 (*Zachowanie po stopie awaryjnym*)
 IF P00_Alarms.aLastStationsErrors[1].nErrorCode >= 1 AND P00_Alarms.aLastStationsErrors[1].nErrorCode <= 20 THEN
     //Jezeli było w trakcie dozowania i coś wydozowało
     IF (iDispencersCase = 4 ) OR (lrDosedMass1CVAux>2 OR lrDosedMass2CVAux>2 OR lrDosedMass3CVAux>2 OR lrDosedMass4CVAux > 2) THEN
         eDispencersPackageState[4].bDoseAborted:=TRUE;
         eDispencersPackageState[3].bDoseAborted:=TRUE;
         eDispencersPackageState[2].bDoseAborted:=TRUE;
         eDispencersPackageState[1].bDoseAborted:=TRUE;
     END_IF
 END_IF
 (*Zachowanie po jakimkolwiek błędzie dozownika 1 i dozownika 2*)
 IF P00_Alarms.aLastStationsErrors[9].bError OR P00_Alarms.aLastStationsErrors[10].bError OR P00_Alarms.aLastStationsErrors[11].bError OR P00_Alarms.aLastStationsErrors[12].bError  THEN
     //Jezeli było w trakcie dozowania i coś wydozowało
     IF (iDispencersCase = 4 ) OR (ABS(lrDosedMass1CVAux)>2 OR ABS(lrDosedMass2CVAux)>2 OR ABS(lrDosedMass3CVAux)>2 OR ABS(lrDosedMass4CVAux) > 2) THEN
         eDispencersPackageState[4].bDoseAborted:=TRUE;
         eDispencersPackageState[3].bDoseAborted:=TRUE;
         eDispencersPackageState[2].bDoseAborted:=TRUE;
         eDispencersPackageState[1].bDoseAborted:=TRUE;
     END_IF
 END_IF
  (*Zachowanie po błędzie przeciagania*)
 IF P00_Alarms.aLastStationsErrors[4].bError OR P00_Alarms.aLastStationsErrors[41].bError OR (P00_Alarms.aLastStationsErrors[1].bError AND P00_Alarms.aLastStationsErrors[1].nErrorCode=70)THEN //Prawe/Lewe
         eBeforeDispencersPackageState[4].bDoseAborted:=TRUE;
         eBeforeDispencersPackageState[3].bDoseAborted:=TRUE;
         eBeforeDispencersPackageState[2].bDoseAborted:=TRUE;
         eBeforeDispencersPackageState[1].bDoseAborted:=TRUE;
     	 eDispencersPackageState[4].bDoseAborted:=TRUE;
         eDispencersPackageState[3].bDoseAborted:=TRUE;
         eDispencersPackageState[2].bDoseAborted:=TRUE;
         eDispencersPackageState[1].bDoseAborted:=TRUE;		  
 END_IF
 
(*Zachowanie po błędzie sortera nasadek*)
 IF P00_Alarms.aLastStationsErrors[50].bError THEN
	
		iCapSorterCase := 0;
		eCapSorterPackageState[1].bCapSorterPuttedAborted	:=	TRUE;
		eCapSorterPackageState[2].bCapSorterPuttedAborted	:=	TRUE;
		eCapSorterPackageState[3].bCapSorterPuttedAborted	:=	TRUE;
		eCapSorterPackageState[4].bCapSorterPuttedAborted	:=	TRUE;
	
 END_IF
 
 (*
 (*Zachowanie po błędzie przeciągania sortera nasadek*)	(*Błąd zablokowanej nasadki*)
 IF P00_Alarms.aLastStationsErrors[51].bError OR (P00_Alarms.aLastStationsErrors[1].bError AND P00_Alarms.aLastStationsErrors[1].nErrorCode=64) THEN
	
		eCapSorterPackageState[1].bCapSorterPuttedAborted	:=	TRUE;
		eCapSorterPackageState[2].bCapSorterPuttedAborted	:=	TRUE;
		eCapSorterPackageState[3].bCapSorterPuttedAborted	:=	TRUE;
		eCapSorterPackageState[4].bCapSorterPuttedAborted	:=	TRUE;

		eBeforeCapSorterPackageState[1].bCapSorterPuttedAborted	:=	TRUE;
		eBeforeCapSorterPackageState[2].bCapSorterPuttedAborted	:=	TRUE;
		eBeforeCapSorterPackageState[3].bCapSorterPuttedAborted	:=	TRUE;
		eBeforeCapSorterPackageState[4].bCapSorterPuttedAborted	:=	TRUE;
	
 END_IF
 *)
END_ACTION

ACTION ACT_ResetAfterStart:
	IF rtResetAfterStart.Q THEN //po 60s
		
		GVL.eCapSorterPackageState[1] 				:= GVL.eClearPackageState;
		GVL.eCapSorterPackageState[2] 				:= GVL.eClearPackageState;
		GVL.eCapSorterPackageState[3] 				:= GVL.eClearPackageState;
		GVL.eCapSorterPackageState[4] 				:= GVL.eClearPackageState;	
	
		GVL.eBeforeCapSorterPackageState[1] 		:= GVL.eClearPackageState;
		GVL.eBeforeCapSorterPackageState[2] 		:= GVL.eClearPackageState;
		GVL.eBeforeCapSorterPackageState[3] 		:= GVL.eClearPackageState;
		GVL.eBeforeCapSorterPackageState[4] 		:= GVL.eClearPackageState;
	
		GVL.eWeightPackageState[1] 					:= GVL.eClearPackageState;
		GVL.eWeightPackageState[2] 					:= GVL.eClearPackageState;
		GVL.eWeightPackageState[3] 					:= GVL.eClearPackageState;
		GVL.eWeightPackageState[4] 					:= GVL.eClearPackageState;

		GVL.eAfterDispencersPackageState[1]			:= GVL.eClearPackageState;
		GVL.eAfterDispencersPackageState[2]			:= GVL.eClearPackageState;
		GVL.eAfterDispencersPackageState[3]			:= GVL.eClearPackageState;	
		GVL.eAfterDispencersPackageState[4]			:= GVL.eClearPackageState;	
	
	
		eBeforeLidFeeder2PackageState[4]			:= GVL.eClearPackageState;		
		eBeforeLidFeeder2PackageState[3]			:= GVL.eClearPackageState;	
		eBeforeLidFeeder2PackageState[2]			:= GVL.eClearPackageState;	
		eBeforeLidFeeder2PackageState[1]			:= GVL.eClearPackageState;	
			
		eBeforeLidFeederPackageState[2]				:= GVL.eClearPackageState;		
		eBeforeLidFeederPackageState[1]				:= GVL.eClearPackageState;		
				
		eLidFeederPackageState[2]					:= GVL.eClearPackageState;		
		eLidFeederPackageState[1]					:= GVL.eClearPackageState;		
				
		eAfterLidFeederPackageState[2]				:= GVL.eClearPackageState;	
		eAfterLidFeederPackageState[1]				:= GVL.eClearPackageState;		
				
		eBeforeLidSealerPackageState[2]				:= GVL.eClearPackageState;		
		eBeforeLidSealerPackageState[1]				:= GVL.eClearPackageState;		
				
		eLidSealerPackageState[2]					:= GVL.eClearPackageState;	
		eLidSealerPackageState[1]					:= GVL.eClearPackageState;	
		
		(*Ustawianie licznika zależnie od czujnika*)
		//IF fbIbCapPuttedCheckFormSensor.bOUT THEN	//Czujnik 5 formatki przed zakrecarkami 
		//	VIS.iNumbersOfFormsBetweenWeightAndScrewers := 1;
		//ELSE
			VIS.iNumbersOfFormsBetweenWeightAndScrewers := 0;
		//END_IF
		irtResetAfterStart	:=	irtResetAfterStart	+	1;
	END_IF
END_ACTION

ACTION ACT_ResetCommands:
(*Resetowanie wszystkich rozkazów*)
(*Zachować kolejność stacji*)



ACT_ResetCommandsHoming();

//Czy na pewno kasowac?
//VIS.bMachinePartsChangeover				:=FALSE;

VIS.bAllowStart:=FALSE;
VIS.bCheckStart:=FALSE;
VIS.bRecipeLoading:=FALSE;

VIS.bCapSorterEmptyingMode				:= FALSE;		
VIS.bBottleSorterEmptyingMode			:= FALSE;	
bCapSorterBottleSorterAutoStart			:= FALSE;
P06_LidSealer.bMovetoEndPositionLidSealer	:=FALSE;
P06_LidFeeder.bMovetoEndPositionLidFeeder	:=FALSE;
(********** Pack_ML*************)
//iStoppingCase							:= 0;
bDelayAfterStart						:= FALSE;
iWeightCase								:= 0;
brtLongDelayFirstDraging				:= FALSE;
bFirstDragingWickFeederAfterRestart1	:= FALSE;
bFirstDragingLidFeederAfterRestart1		:= FALSE;
bFirstDragingLidFeederAfterRestart2		:= FALSE;
bFirstDragingLidSealerAfterRestart1		:= FALSE;
bFirstDragingLidSealerAfterRestart2		:= FALSE;
iFirstDragingLidFeederAfterRestart2Count:=0;
iFirstDragingLidSealerAfterRestart2Count:=0;

//bBottleFeederHommed					:=FALSE;
//bFormsDragRightStationHommed			:=FALSE;
//bFormsDragLeftStationHommed			:=FALSE;
//bDispencersHommed    					:=FALSE; 
//bWeightLiftHommed		                :=FALSE; 
//bCapFeederHommed 						:=FALSE;
//bCapPuttedCheckHommed	                :=FALSE; 
//bBottleDragHommed		                :=FALSE; 
//bGripperScrewerHommed                 :=FALSE; 
//bCapSorterDragHommed					:=FALSE;
//bCapCorrectCheckHommed                :=FALSE; 
//bBottleTransferHommed	                :=FALSE; 


(** P01_BottleFeeder***)
//bBottleFeederDoHoming					:=FALSE;
//VIS.bBottleFeederHoming				:=FALSE;
bBottleFeederFormGateRun				:=FALSE;
bBottleFeederTurnTableRun				:=FALSE;
VIS.bBottleFeederRun					:=FALSE;
///////////////////////// dodane bo nie było
VIS.bBottleFeederManualArmDown			:=FALSE;
VIS.bBottleFeederManualArmLeft			:=FALSE;
VIS.bBottleFeederManualFormGate			:=FALSE;
VIS.bBottleFeederManualGate1			:=FALSE;
VIS.bBottleFeederManualGate2			:=FALSE;
VIS.bBottleFeederManualGripper			:=FALSE;
VIS.bBottleFeederManualFormPositioning	:=FALSE;
VIS.bBottleFeederTurnTableManualCmdStart:=FALSE;
///////////////////////

(** P01_PucksInserter***)
//bPucksInserterDoHoming				:=FALSE;
//VIS.bPucksInserterHoming				:=FALSE;
bPucksInserterFormGateRun				:=FALSE;
bPucksInserterTurnTableRun				:=FALSE;
VIS.bPucksInserterRun					:=FALSE;
VIS.bPucksInserterManualHammer			:=FALSE;								
//VIS.bPucksInserterManualTray			:=FALSE;								
//VIS.bPucksInserterManualGate1			:=FALSE;								
//IS.bPucksInserterManualGate2			:=FALSE;								
VIS.bPucksInserterManualFormGate		:=FALSE;								
VIS.bPucksInserterManualFormPositioning	:=FALSE;								
VIS.bPucksInserterManualWheelLeft		:=FALSE;
VIS.bPucksInserterManualWheelRight		:=FALSE;
VIS.bPucksInserterConveyorManualCmdStart:=FALSE;								
VIS.bPucksInserterManualHammerUp		:=FALSE;
VIS.bPucksInserterManualHammerDown		:=FALSE;
VIS.bPucksInserterTurnTableManualCmdStart:=FALSE;
//Vasyl 27.05
bPucksInserterPushTable_m1_Run			:=FALSE;
bPucksInserterPushTable_m2_Run			:=FALSE;
bPucksInserterPushTable_m3_Run			:=FALSE;
///////////////////////

//Gates
//VIS.bGateBeforeWeight14Run			:= FALSE;
//VIS.bGateBeforeWeight56Run			:= FALSE;
VIS.bGateRobotEntranceRun				:= FALSE;	
VIS.bGateBeforeDispencersRun			:= FALSE;

(******* P02_Dispencers ********)
bFormsDragingRightPrepareRun			:=FALSE;
VIS.bFormsDragingRightRun 				:=FALSE;
//VIS.bFormsDragingRightHoming			:=FALSE;
//bFormsDragingRightDoHoming			:=FALSE;
//bFormsDragingRightHeightSet			:=FALSE;
VIS.bFormsDragingRightManualFork		:=FALSE;	
VIS.bFormsDragingRightManualLeadBefore1	:=FALSE;	
VIS.bFormsDragingRightManualLeadBefore2	:=FALSE;	
VIS.bFormsDragingRightManualLeft		:=FALSE;							
VIS.bFormsDragingRightManualRight		:=FALSE;
bFormsDragingRightRunCheck				:=FALSE;

bFormsDragingLeftPrepareRun				:=FALSE;
VIS.bFormsDragingLeftRun 				:=FALSE;
//VIS.bFormsDragingLeftHoming			:=FALSE;
//bFormsDragingLeftDoHoming				:=FALSE;
//bFormsDragingLeftHeightSet				:=FALSE;
VIS.bFormsDragingLeftManualFork			:=FALSE;	
VIS.bFormsDragingLeftManualLeadBefore1	:=FALSE;	
VIS.bFormsDragingLeftManualLeadBefore2	:=FALSE;												
VIS.bFormsDragingLeftManualLeft			:=FALSE;							
VIS.bFormsDragingLeftManualRight		:=FALSE;
bFormsDragingLeftRunCheck				:=FALSE;

//bDispencersDoHoming					:= FALSE;
//VIS.bDispencersHoming 				:= FALSE;
VIS.bDispencersManualDropCatcher 		:= FALSE;
VIS.bDispencersManualLifterUp			:= FALSE;
VIS.bDispencersManualLifterDown			:= FALSE;

bDispencer1Cleaning	:= FALSE;	
bDispencer2Cleaning	:= FALSE;	
bDispencer3Cleaning	:= FALSE;	
bDispencer4Cleaning	:= FALSE;	

bDispencer1DoSync	:= FALSE;
bDispencer1DoSync	:= FALSE;
bDispencer1DoSync	:= FALSE;
bDispencer1DoSync	:= FALSE;

VIS.bDispencersPullingFast 				:= FALSE;  	
VIS.bDispencersPullingSlow 				:= FALSE;  	
VIS.bDispencersPullingFastContinous		:= FALSE;  	
VIS.bDispencersPullingSlowContinous		:= FALSE;  	
VIS.bDispencersDose						:= FALSE;  

//VIS.bDispencer12LifterHeightSet		:= FALSE;
VIS.bDispencer1Dose        				:= FALSE;
VIS.bDispencer1PullingFast 				:= FALSE;
VIS.bDispencer1PullingSlow 				:= FALSE;

VIS.bDispencer2Dose        				:= FALSE;
VIS.bDispencer2PullingFast 				:= FALSE;
VIS.bDispencer2PullingSlow				:= FALSE;

//VIS.bDispencer34LifterHeightSet		:= FALSE;
VIS.bDispencer3Dose        				:= FALSE;
VIS.bDispencer3PullingFast 				:= FALSE;
VIS.bDispencer3PullingSlow 				:= FALSE;

VIS.bDispencer4Dose        				:= FALSE;
VIS.bDispencer4PullingFast 				:= FALSE;
VIS.bDispencer4PullingSlow 				:= FALSE;

VIS.bDispencer1ManualSuckValve			:= FALSE;
VIS.bDispencer1ManualDoseValve			:= FALSE;
VIS.bDispencer2ManualSuckValve			:= FALSE;
VIS.bDispencer2ManualDoseValve			:= FALSE;
VIS.bDispencer3ManualSuckValve			:= FALSE;
VIS.bDispencer3ManualDoseValve			:= FALSE;
VIS.bDispencer4ManualSuckValve			:= FALSE;
VIS.bDispencer4ManualDoseValve			:= FALSE;
		
VIS.bDispencers1Catch 					:= FALSE;
VIS.bDispencers2Catch 					:= FALSE;
VIS.bDispencers3Catch 					:= FALSE;
VIS.bDispencers4Catch 					:= FALSE;

//VIS.bDispencersCatchHeightSet			:=FALSE;

//bDispencersCatch1DoHoming				:=FALSE;
//bDispencersCatch2DoHoming				:=FALSE;
//bDispencersCatch3DoHoming				:=FALSE;
//bDispencersCatch4DoHoming				:=FALSE;

(*******P05_Weight*******)
VIS.bWeightLiftRun 						:=FALSE;
bWeightLift2PhaseRun					:=FALSE;
bWeightLiftDeparture					:=FALSE;

//VIS.bWeightLiftHoming					:=FALSE;	
//GVL.bWeightLiftDoHoming				:=FALSE;

VIS.bWeight1DoWeighting 				:= FALSE;
VIS.bWeight1Tare        				:= FALSE;
VIS.bWeight2DoWeighting 				:= FALSE;
VIS.bWeight2Tare        				:= FALSE;
VIS.bWeight3DoWeighting 				:= FALSE;
VIS.bWeight3Tare        				:= FALSE;
VIS.bWeight4DoWeighting					:= FALSE;
VIS.bWeight4Tare       					:= FALSE;

VIS.bWeight5DoWeighting 						:= FALSE;
VIS.bWeight5Tare        				:= FALSE;
VIS.bWeight6DoWeighting							:= FALSE;
VIS.bWeight6Tare       					:= FALSE;
/////////////////////////////////// nie było to dodaje
VIS.bWeight1ActuatorManualUp			:=FALSE;
VIS.bWeight1ActuatorManualDown			:=FALSE;
VIS.bWeight2ActuatorManualUp			:=FALSE;
VIS.bWeight2ActuatorManualDown			:=FALSE;
VIS.bWeight3ActuatorManualUp			:=FALSE;
VIS.bWeight3ActuatorManualDown			:=FALSE;
VIS.bWeight4ActuatorManualUp			:=FALSE;
VIS.bWeight4ActuatorManualDown			:=FALSE;
VIS.bWeight5ActuatorManualUp			:=FALSE;
VIS.bWeight5ActuatorManualDown			:=FALSE;
VIS.bWeight6ActuatorManualUp			:=FALSE;
VIS.bWeight6ActuatorManualDown			:=FALSE;
 
(*****P08_CapFeeder********)
VIS.bCapFeederRun:=FALSE;	
VIS.bCapFeederManualHeightUp:=FALSE;	
VIS.bCapFeederManualHeightDown:=FALSE;	
VIS.bCapFeederManualSorterEngine:=FALSE;	
VIS.bCapFeederManualSorterAir:=FALSE;		
VIS.bCapFeederManualGate1:=FALSE;	
VIS.bCapFeederManualGate2:=FALSE;	
//bCapFeederDoHoming:=FALSE;
//VIS.bCapFeederHeightSet:=FALSE;	
iCapFeederCheckCountNOK:=0;

(*****P08_CapFeeder********)
VIS.bWickFeederSorterRun					:=FALSE;
VIS.bWickFeeder1PrepareRun					:=FALSE;
VIS.bWickFeeder1Run							:=FALSE;
VIS.bWickFeeder2PrepareRun					:=FALSE;
VIS.bWickFeeder2Run							:=FALSE;
VIS.bWickFeederManualHeightUp				:=FALSE;
VIS.bWickFeederManualHeightDown				:=FALSE;
VIS.bWickFeederManualSorterEngine			:=FALSE;
VIS.bWickFeederManualSorterAir				:=FALSE;
VIS.bWickFeederManualStopper				:=FALSE;
VIS.bWickFeederManualStopper2				:=FALSE;
VIS.bWickFeederManualSeparator1				:=FALSE;
VIS.bWickFeederManualSeparator2				:=FALSE;
VIS.bWickFeederManualSleve1SeparatorActIn	:=FALSE;
VIS.bWickFeederManualSleve1SeparatorActOut	:=FALSE;
VIS.bWickFeederManualSleve2SeparatorActIn	:=FALSE;
VIS.bWickFeederManualSleve2SeparatorActOut	:=FALSE;
VIS.bWickFeederManualHammer1				:=FALSE;
VIS.bWickFeederManualHammer2				:=FALSE;
VIS.bWickFeederManualFormPositioning		:=FALSE;
//Podawanie knotów - przeciąganie		
VIS.bWickFeederDragingStationRun			:=FALSE;					
bWickFeederDragingStationPrepareRun			:=FALSE;
VIS.bWickFeederDragingManualFork			:=FALSE;
VIS.bWickFeederDragingManualLeadBefore1		:=FALSE;
VIS.bWickFeederDragingManualLeadBefore2		:=FALSE;
VIS.bWickFeederDragingManualLeft			:=FALSE;
VIS.bWickFeederDragingManualRight			:=FALSE;
iWickFeederDragStoppingCount				:=0;

(*****P06_LidFeeder*************)
VIS.bLidFeederManualHeightUp			:=FALSE;	
VIS.bLidFeederManualHeightDown			:=FALSE;	
VIS.bLidFeederManualFormPositioning		:=FALSE;	
VIS.bLidFeederManualFormPositioning		:=FALSE;	
//VIS.bLidFeeder1PrepareRun				:=FALSE;	
VIS.bLidFeeder1Run						:=FALSE;	
VIS.bLidFeeder1ManualAct				:=FALSE;	
VIS.bLidFeeder1ManualAct2				:=FALSE;	
VIS.bLidFeeder1ManualSuckerAct			:=FALSE;	
VIS.bLidFeeder1ManualHeaterAct			:=FALSE;
bLidFeederFormPositioningRun			:=FALSE;
//VIS.bLidFeeder2PrepareRun				:=FALSE;
VIS.bLidFeeder2Run						:=FALSE;	
VIS.bLidFeeder2ManualAct				:=FALSE;	
VIS.bLidFeeder2ManualAct2				:=FALSE;	
VIS.bLidFeeder2ManualSuckerAct			:=FALSE;	
VIS.bLidFeeder2ManualHeaterAct			:=FALSE;	
VIS.bLidFeederDragingStationRun			:=FALSE;
VIS.bLidFeederDragingManualFork			:=FALSE; 
VIS.bLidFeederDragingManualLeadBefore1	:=FALSE; 
VIS.bLidFeederDragingManualLeadBefore2	:=FALSE; 
VIS.bLidFeederDragingManualLeft			:=FALSE;
VIS.bLidFeederDragingManualRight		:=FALSE;
iLidFeederDragStoppingCount				:=0;
	
(*****P06_LidPuttedCheck********)
VIS.bLidPuttedCheckRun					:=FALSE;	
VIS.bLidPuttedCheckManualHeightUp  	 	:=FALSE;	
VIS.bLidPuttedCheckManualHeightDown	 	:=FALSE;	

(*****P06_LidSealer************)
VIS.bLidSealerManualHeightUp			:=FALSE;		
VIS.bLidSealerManualHeightDown  		:=FALSE;	
VIS.bLidSealer1Run              		:=FALSE;	
VIS.bLidSealer1ManualAct        		:=FALSE;		
VIS.bLidSealer2Run              		:=FALSE;	
VIS.bLidSealer2ManualAct        		:=FALSE;	
VIS.bLidSealerDragingStationRun			:=FALSE;	
VIS.bLidSealerDragingManualFork			:=FALSE;		
VIS.bLidSealerDragingManualLeadBefore1	:=FALSE;	
VIS.bLidSealerDragingManualLeadBefore2	:=FALSE;	
VIS.bLidSealerDragingManualLeft			:=FALSE;		
VIS.bLidSealerDragingManualRight		:=FALSE;	
iLidSealerDragStoppingCount				:=0;

(*****P07_CapPusher********)

iCapPusherGateCase								:= 0;	
iCapPusherCase									:= 0;	
bCapPusherGateRun								:= FALSE;
bCapPusherManualGate							:= FALSE;

VIS_CP.bCapPusherFeederRun						:= FALSE;
VIS_CP.bCapPusherFeederHeightSet				:= FALSE;
VIS_CP.bCapPusherFeederManualSorterEngine		:= FALSE;
VIS_CP.bCapPusherFeederManualSorterVibrator	    := FALSE;
VIS_CP.bCapPusherFeederManualSorterVibrator2	:= FALSE;
VIS_CP.bCapPusherFeederManualSorterAir			:= FALSE;

VIS_CP.bCapPusherRun							:= FALSE;
VIS_CP.bCapPusherHeightSet				        := FALSE;
VIS_CP.bCapPusherManualPusher			        := FALSE;
VIS_CP.bCapPusherManualBlockActuator	        := FALSE;
VIS_CP.bCapPusherManualFormPositioning	        := FALSE;

(*****P07_ROPP********)
//Spowalniacz
bROPPSlowerCmdStart						:=	FALSE;
VIS_ROPP.bROPPSlowerManualCmdStart		:=	FALSE;

//Podajnik 
VIS_ROPP.bROPPFeederRun					:=	FALSE;					
VIS_ROPP.bROPPFeederManualHeightUp		:=	FALSE;		
VIS_ROPP.bROPPFeederManualHeightDown	:=	FALSE;		
VIS_ROPP.bROPPFeederManualSorterEngine	:=	FALSE;		
VIS_ROPP.bROPPFeederManualSorterVibrator:=	FALSE;		
VIS_ROPP.bROPPFeederManualSorterAir		:=	FALSE;			
VIS_ROPP.bROPPFeederManualSorterAir2	:=	FALSE;			
VIS_ROPP.bROPPFeederManualConveyorStart	:=	FALSE;		
VIS_ROPP.bROPPFeederManualConveyorStop	:=	FALSE;		
//Sprawdzanie kapsla
iROPPFeederCheckCountNOK				:= 0;

//Przeciąganie formatek 
bROPPDragPrepareRun						:=	FALSE;
VIS_ROPP.bROPPDragRun					:=	FALSE;
VIS_ROPP.bROPPDragManualFork			:=	FALSE;	
VIS_ROPP.bROPPDragManualLead			:=	FALSE;	
VIS_ROPP.bROPPDragManualLeft			:=	FALSE;	
VIS_ROPP.bROPPDragManualRight			:=	FALSE;
//Zakrecanie
bROPPCappingRunEngine									:=	FALSE;
VIS_ROPP.bROPPCappingRun1								:=	FALSE;					
VIS_ROPP.bROPPCappingRun2								:=	FALSE;										
VIS_ROPP.bROPPCappingManualHeightUp						:=	FALSE;				
VIS_ROPP.bROPPCappingManualHeightDown					:=	FALSE;				
VIS_ROPP.bROPPCappingManualEngine1						:=	FALSE;				
VIS_ROPP.bROPPCappingManualEngine2						:=	FALSE;					
VIS_ROPP.bROPPCappingManualCapping1Tool1Actuator		:=	FALSE;		
VIS_ROPP.bROPPCappingManualCapping2Tool1Actuator		:=	FALSE;		
VIS_ROPP.bROPPCappingManualCapping12Tool1BlockActuator	:=	FALSE;
VIS_ROPP.bROPPCappingManualCappingBlockActuator			:=	FALSE;	
VIS_ROPP.bROPPCappingManualCapping1Tool2Down			:=	FALSE;			
VIS_ROPP.bROPPCappingManualCapping1Tool2Tight			:=	FALSE;		
VIS_ROPP.bROPPCappingManualCapping1Tool2Realese			:=	FALSE;		
VIS_ROPP.bROPPCappingManualCapping2Tool2Down			:=	FALSE;			
VIS_ROPP.bROPPCappingManualCapping2Tool2Tight			:=	FALSE;		
VIS_ROPP.bROPPCappingManualCapping2Tool2Realese			:=	FALSE;		
VIS_ROPP.bROPPCappingManualFormPositioning				:=	FALSE;			
//Sprawdzanie kapsla 	


(*****P08_CapSorter********)
bCapSorterDragPrepareRun				:=FALSE;
VIS.bCapSorterDragRun 					:=FALSE;
///VIS.bCapSorterDragHoming				:=FALSE;
//bCapSorterDragDoHoming				:=FALSE;
//bCapSorterDragHeightSet				:=FALSE;
VIS.bCapSorterDragManualFork			:=FALSE;	
VIS.bCapSorterDragManualLeadBefore1		:=FALSE;	
VIS.bCapSorterDragManualLeft			:=FALSE;							
VIS.bCapSorterDragManualRight			:=FALSE;
 
//iCapSorterCase							:=0;
bCapSorterRobotPlace					:=FALSE;			
bCapSorterRobotBottleAndNoCap1			:=FALSE;
bCapSorterRobotBottleAndNoCap2			:=FALSE;	
bCapSorterRobotBottleAndNoCap3			:=FALSE;	
bCapSorterRobotBottleAndNoCap4			:=FALSE;	
bCapSorterRobotPreparePlace				:=FALSE;	
bCapSorterBeforeRobotBottleAndNoCap1	:=FALSE;	
bCapSorterBeforeRobotBottleAndNoCap2	:=FALSE;	
bCapSorterBeforeRobotBottleAndNoCap3	:=FALSE;	
bCapSorterBeforeRobotBottleAndNoCap4	:=FALSE;	
bCapSorterError							:=FALSE;

(*****P09_CapPuttedCheck********)
bCapPuttedCheckRun						:=FALSE;
//VIS.bCapPuttedCheckHoming				:=FALSE;
VIS.bCapPuttedCheckManualHeightUp		:=FALSE; 								// Ręczne podnoszenie stacji sprawdzania nasadek
VIS.bCapPuttedCheckManualHeightDown		:=FALSE;			 					// Reczne opuszczanie stacji sprawdzania nasadek
//VIS.bCapPuttedCheckHeightSet			:=FALSE;
//bCapPuttedCheckDoHoming				:=FALSE;

(*****P10_GripperScrewer********)
(*** Przeciąganie formatek z butlekmami****)
VIS.bBottleDragingStationRun			:=FALSE;
GVL.bBottleDragingStationPrepareRun		:=FALSE;
VIS.bBottleDragingStationManualFork1	:=FALSE;
VIS.bBottleDragingStationManualLead		:=FALSE;
VIS.bBottleDragingStationManualLeft		:=FALSE;
VIS.bBottleDragingStationManualRight	:=FALSE;
//VIS.bBottleDragingStationHoming		:=FALSE;
//bBottleDragingStationDoHoming			:=FALSE;
//bBottleDragingHeightSet				:=FALSE;

(*****P10_GripperScrewer********)
//VIS.bGripperScrewerHoming				:=FALSE; 
VIS.bGripperScrewer1Run					:=FALSE;
VIS.bGripperScrewerLiftManualHeightUp	:=FALSE;
VIS.bGripperScrewerLiftManualHeightDown	:=FALSE;
VIS.bGripperScrewer1ManualRight			:=FALSE;			
VIS.bGripperScrewer1ManualLeft			:=FALSE;
VIS.bGripperScrewer1ManualCatch			:=FALSE;
//VIS.bGripperScrewerHeightSet			:=FALSE;
VIS.bGripperScrewer1AdjustTorque		:=FALSE;
//bGripperScrewerDoHoming				:=FALSE;

VIS.bGripperScrewer2Run					:=FALSE;
VIS.bGripperScrewer2ManualRight			:=FALSE;			
VIS.bGripperScrewer2ManualLeft			:=FALSE;
VIS.bGripperScrewer2ManualCatch			:=FALSE;

(*** Chwytak butelek***)
//VIS.bGripperScrewerCatchHeightSet		:=FALSE;
VIS.bGripperScrewerCatchManualUp		:=FALSE;
VIS.bGripperScrewerCatchManualDown		:=FALSE;
//GVL.bGripperScrewerCatch1Homing		:=FALSE;
//GVL.bGripperScrewerCatch2Homing		:=FALSE;
//bGripperScrewerCatch1DoHoming			:=FALSE;
//bGripperScrewerCatch2DoHoming			:=FALSE;
bGripperScrewer1Catch 					:=FALSE;
bGripperScrewer2Catch 					:=FALSE;
VIS.bGripperScrewerCatch2ManualActuator	:=FALSE;
VIS.bGripperScrewerCatch1ManualActuator	:=FALSE;

(*****P09_CapCorrectCheck********)
//VIS.bCapCorrectCheckHoming         	:= FALSE;
//bCapCorrectCheckDoHoming        		:= FALSE;
VIS.bCapCorrectCheckHeightSet       	:= FALSE;
VIS.bCapCorrectCheckManualHeightUp  	:= FALSE;
VIS.bCapCorrectCheckManualHeightDown 	:= FALSE;
//bCapCorrectCheckDoHoming				:=FALSE;

//ROBOT
VIS.bBottleTransferRun					:=FALSE;
//VIS.bBottleTransferHoming				:=FALSE;
VIS.bBottleTransferPlace				:=FALSE;
VIS.bBottleTransferManualEditOffset		:=FALSE;
VIS.bBottleTransferManualPick			:=FALSE;
VIS.bBottleTransferManualPick2			:=FALSE;
VIS.bBottleTransferManualPlace1			:=FALSE;
VIS.bBottleTransferManualPlace2			:=FALSE;
VIS.bBottleTransferManualReadyPosition	:=FALSE;
VIS.bBottleTransferManualStartInkJet	:=FALSE;
VIS.bBottleTransferManualStopInkJet		:=FALSE;
VIS.bBottleTransferManualWeight			:=FALSE;
VIS.bBottleTransferManualCatch			:=FALSE;

(*****P13_BottleTransferAfterDrag********)
VIS.bBottleTransferAfterDragRun				:=FALSE;
VIS.bBottleTransferAfterDragManualActuator	:=FALSE;
VIS.bBottleTransferAfterDragManualStoper	:=FALSE;	
VIS.bBottleTransferAfterDragManualGate		:=FALSE;	


(***** P15_FormTransporter*******)
VIS.bFormTransporterDispencerManualCmdStart 	:=FALSE;
VIS.bFormTransporterScrewerManualCmdStart 		:=FALSE;
VIS.bFormTransporterBeforeScrewerManualCmdStart :=FALSE;
VIS.bFormTransporterAfterCapSorterManualCmdStart :=FALSE;
VIS.bBadBottleConveyorManualCmdStart			:=FALSE;

bFormTransportersDispencerCmdStart		 := FALSE;
bFormTransportersScrewerCmdStart		 := FALSE;
bFormTransportersScrewerStop 			 := FALSE;
//bFormTransportersScrewerSlow			 := FALSE; //Nie dodawać do ResetCommands
bFormTransportersAfterCapSorterCmdStart	 := FALSE;
bFormTransportersBeforeScrewerCmdStart	 := FALSE;
bFormTransportersAfterScrewerCmdStart	 := FALSE;
QbBlowAfterGripperScrewer				 := FALSE;
QbBlowBeforeGripperScrewer				 := FALSE;
iGateBeforeGripperScrewerCase			 :=	0;


VIS.bLabelMachine1ManualStart			:= FALSE;
	bLabelMachineCmdStart 				:= FALSE;	


//bExitTurnTableCmdStart	:= FALSE;
VIS.bExitTurnTable1ManualStart:= FALSE;
//bExitConveyorCmdStart	:= FALSE;	
	
(*P20_Exhaust*)
VIS.bExhaustFanManualCmdStart		:= FALSE;
END_ACTION

ACTION ACT_ResetCommandsHoming:

IF NOT (fbPMLModeManager.eModeStatus = Tc3_PackML.E_PMLUnitMode.ePMLUnitMode_MANUAL) OR  (fbPMLAuto.ePMLState=Tc3_PackML.E_PMLState.ePMLState_ABORTING OR fbPMLManual.ePMLState=Tc3_PackML.E_PMLState.ePMLState_ABORTING) THEN
	
	//bRecipeChangePositioning						:=FALSE;
	
	bHoming											:=FALSE;
	iHomingCase										:=0;

	bBottleFeederDoHoming							:=FALSE;
	VIS.bBottleFeederHoming							:=FALSE;
	bPucksInserterDoHoming							:=FALSE;
	VIS.bPucksInserterHoming						:=FALSE;
	VIS.bPucksInserterHeightSet						:=FALSE;
	
	GvlCommunication.stBottleSorterWrite.bHoming	:=FALSE;
	
	VIS.bFormsDragingRightHoming					:=FALSE;
	bFormsDragingRightDoHoming						:=FALSE;
	bFormsDragingRightHeightSet						:=FALSE;
	VIS.bFormsDragingLeftHoming						:=FALSE;
	bFormsDragingLeftDoHoming						:=FALSE;
	bFormsDragingLeftHeightSet						:=FALSE;
	bDispencersDoHoming								:=FALSE;	
	VIS.bDispencersHoming 							:=FALSE;	
	VIS.bDispencersCatchHeightSet					:=FALSE;	
	VIS.bDispencer12LifterHeightSet					:= FALSE;	
	VIS.bDispencer34LifterHeightSet					:= FALSE;	
	bDispencersCatch1DoHoming						:=FALSE;
	bDispencersCatch2DoHoming						:=FALSE;
	bDispencersCatch3DoHoming						:=FALSE;
	bDispencersCatch4DoHoming						:=FALSE;	
	VIS.bWeightLiftHoming							:=FALSE;	
	GVL.bWeightLiftDoHoming							:=FALSE;	
	
	VIS.bWickFeederHoming							:=FALSE;
	bWickFeederDoHoming								:=FALSE;
	VIS.bWickFeederHeightSet						:=FALSE;
	VIS.bWickFeederDragingHoming					:=FALSE;
	bWickFeederDragingStationDoHoming				:=FALSE;
	
	VIS.bLidFeederHoming							:=FALSE;
	VIS.bLidFeederHeightSet							:=FALSE;
	GVL.bLidFeederDoHoming							:=FALSE;
	VIS.bLidFeederDragingHoming						:=FALSE;
	GVL.bLidFeederDragingStationDoHoming			:=FALSE;
	VIS.bLidPuttedCheckHoming						:=FALSE;
	VIS.bLidPuttedCheckHeightSet					:=FALSE;
	GVL.bLidPuttedCheckDoHoming						:=FALSE;
	VIS.bLidSealerHoming							:=FALSE;
	VIS.bLidSealerHeightSet							:=FALSE;
	GVL.bLidSealerDoHoming							:=FALSE;
	VIS.bLidSealerDragingHoming						:=FALSE;
	GVL.bLidSealerDragingStationDoHoming			:=FALSE;
	
	//ROPP
	bROPPFeederDoHoming								:=FALSE;
	VIS_ROPP.bROPPFeederHoming						:=FALSE;
	VIS_ROPP.bROPPFeederHeightSet					:=FALSE;
	bROPPDragDoHoming								:=FALSE;
	VIS_ROPP.bROPPDragHoming						:=FALSE;
	bROPPCappingDoHoming							:=FALSE;
	VIS_ROPP.bROPPCappingHoming						:=FALSE;
	VIS_ROPP.bROPPCappingHeightSet					:=FALSE;
	
	bCapFeederDoHoming								:=FALSE;
	VIS.bCapFeederHeightSet							:=FALSE;		
	VIS.bCapSorterDragHoming						:=FALSE;
	bCapSorterDragDoHoming							:=FALSE;
	bCapSorterDragHeightSet							:=FALSE;	
	
	GvlCommunication.stCapSorterWrite.bHoming		:=FALSE;
	
	VIS.bCapPuttedCheckHoming						:=FALSE;
	bCapPuttedCheckDoHoming							:=FALSE;
	VIS.bCapPuttedCheckHeightSet					:=FALSE;
	VIS.bBottleDragingStationHoming					:=FALSE;
	bBottleDragingStationDoHoming					:=FALSE;
	bBottleDragingHeightSet							:=FALSE;
	VIS.bGripperScrewerHoming						:=FALSE; 
	VIS.bGripperScrewerHeightSet					:=FALSE;
	bGripperScrewerDoHoming							:=FALSE;
	VIS.bGripperScrewerCatchHeightSet				:=FALSE;
	GVL.bGripperScrewerCatch1Homing					:=FALSE;
	GVL.bGripperScrewerCatch2Homing					:=FALSE;
	bGripperScrewerCatch1DoHoming					:=FALSE;
	bGripperScrewerCatch2DoHoming					:=FALSE;
	VIS.bCapCorrectCheckHoming         				:=FALSE;
	bCapCorrectCheckDoHoming        				:=FALSE;
	VIS.bCapCorrectCheckHeightSet       			:=FALSE;
	VIS.bBottleTransferHoming						:=FALSE;	
	VIS.bBottleTransferAfterDragHoming				:=FALSE;
	bBottleTransferAfterDragHeightSet				:=FALSE;
	bBottleTransferAfterDragDoHoming				:=FALSE;
	bBottleFeederHommed								:=FALSE;
	bPucksInserterHommed							:=FALSE;	
	bFormsDragRightStationHommed					:=FALSE;
	bFormsDragLeftStationHommed						:=FALSE;
	bDispencersHommed    							:=FALSE; 
	bWeightLiftHommed		        				:=FALSE; 
	bCapFeederHommed 								:=FALSE;
	bCapPuttedCheckHommed	            			:=FALSE; 
	bBottleDragHommed		        				:=FALSE; 
	bGripperScrewerHommed               			:=FALSE; 
	bWickFeederHommed		             			:=FALSE; 	
	bWickFeederDragingHommed	             		:=FALSE; 	
	bLidFeederHommed		             			:=FALSE; 	
	bLidFeederDragingHommed	             			:=FALSE; 	
	bLidPuttedCheckHommed	             			:=FALSE; 	
	bLidSealerHommed		             			:=FALSE; 	
	bLidSealerDragingHommed	             			:=FALSE; 	
	bROPPFeederHommed								:=FALSE; 	
	bROPPDragHommed									:=FALSE; 	
	bROPPCappingHommed								:=FALSE; 	
	bCapSorterDragHommed							:=FALSE;
	bCapCorrectCheckHommed              			:=FALSE; 
	bBottleTransferHommed	            			:=FALSE; 
	bBottleTransferAfterDragHommed					:=FALSE;
END_IF
END_ACTION

ACTION ACT_Resetting:

//1. Przy pierwszym uruchomieniu wszystkie stację się bazują
//2. Bazowania zostają włączone od Enablów lub Not HomingDone, zależnie od miejsca
//3. Gdy wszystkie bazowania zostaną wyłączone w PositioningLogic i okienko zostanie wyłączone to przejdz dalej

// Przejście z Manual-Idle do Resseting jeżeli włączone zostanie któreś bazowanie
// Przejśćie z Automatic-Idle do Resseting jeżeli coś wymaga bazownaia
// Przejśćie z Automatic-Idle jeżeli ktoś wybral nowa recepture z wizki

ftHomingDialog.CLK	:= bHomingDialog;
ftHomingDialog();

IF ftHomingDialog.Q THEN
	iHomingCase		:= 0;
END_IF



//Homing
ACT_HomingCycle();

//Przejdź dalej jeżeli nie jest włączone bazowanie i nie ma błędu
IF (NOT VIS.bErrorOccure AND NOT bHoming AND NOT bHomingDialog) (*OR (GvlVisualization.bServiceMode AND NOT1*) THEN
	
	IF bResetAfterErrorOrEstop THEN //Sprawdzanie czy był błąd podczas ruchu i ustawianie rejestrów
		ACT_ResetAfterErrorOrEstop_do_usun();
		bResetAfterErrorOrEstop := FALSE;
	END_IF

	fbPMLAuto.StateComplete						:= TRUE; 
	fbPMLManual.StateComplete					:= TRUE;
END_IF
END_ACTION

ACTION ACT_SafetyFirstResetDelay:
(*
Nazwa:			ACT_SafetyFirstResetDelay
Opis:			Opóźnienie przy pierwszym resetowaniu safety
Wersja:			v0.1
Data:			2024-06-26
Autor:			DP
Urzadzenia:		
Konfiguracja:	
Info:
- opóżnienie przed pierwszym resetem safety bo robot/ sorter butelek nie wstaje tak szybko
*)
IF bBottleSorterDisable AND bCapSorterDisable OR bSafetyTest THEN
	tonbFirstCycle(IN:=bFirstCycle,PT:=T#10S);
ELSE
	tonbFirstCycle(IN:=bFirstCycle,PT:=T#150S); 	
END_IF
IF tonbFirstCycle.Q THEN 
	QbSafetyResetDelay	:=	TRUE;
END_IF
END_ACTION

ACTION ACT_Signals:
//Dodane oszukiwanie czujnikow ktorych nie ma na maszynie

//MAIN.IbSecondFormCheckFormSensor		:= MAIN.IbFourthFormCheckFormSensor; 




(*Filtr zmiennej ekranu serwisowego*)
fbServiceMode	(bIn:=VIS.bServiceMode,		tFilterTimeOn:=T#1S, tFilterTimeOff:=T#1S);
fbServiceMode.bOut;


rttonDelayAfterStart		(CLK:=tonDelayAfterStart.Q																			,Q=>); 
IF GVL.nFormTransportersBeforeScrewerVelocitySV<1000 THEN
tonDelayAfterStart			(IN := bDelayAfterStart, 																			PT := T#3S);	//Opóźnienie po uruchomieniu cyklu
ELSE
tonDelayAfterStart			(IN := bDelayAfterStart, 																			PT := T#3S);	//Opóźnienie po uruchomieniu cyklu
END_IF
tonDelayAfterStart6s		(IN := bDelayAfterStart, 																			PT := T#6S);	//Opóźnienie po uruchomieniu cyklu


IF bFastSpeed THEN
	tonLongDelayAfterStart.Q;				tonLongDelayAfterStart		(IN := bLongDelayAfterStart, 																		PT := T#40S);	//Opóźnienie po uruchomieniu cyklu
ELSE
	tonLongDelayAfterStart.Q;				tonLongDelayAfterStart		(IN := bLongDelayAfterStart, 																		PT := T#40S);	//Opóźnienie po uruchomieniu cyklu	
END_IF
tonLongDelayAfterStart.ET;
tonLongDelayFirstDraging.Q;				tonLongDelayFirstDraging			(IN := bLongDelayAfterStart,																PT := (tonLongDelayAfterStart.PT / 3));	  //20s
tonLongDelayFirstDragingLidFeeder.Q;	tonLongDelayFirstDragingLidFeeder	(IN := bLongDelayAfterStart,																PT := T#46S); //46s
tonLongDelayFirstDragingLidSealer.Q;	tonLongDelayFirstDragingLidSealer	(IN := bLongDelayAfterStart,																PT := T#54S); //54s

tonStarting.Q;							tonStarting					(IN := fbPMLAuto.ePMLState = Tc3_PackML.E_PMLState.ePMLState_STARTING, 								PT := T#1S500MS);
tonExecute.Q;							tonExecute					(IN := fbPMLAuto.ePMLState = Tc3_PackML.E_PMLState.ePMLState_EXECUTE, 								PT := T#5S);
tonNotExecute.Q;						tonNotExecute				(IN := fbPMLAuto.ePMLState <> Tc3_PackML.E_PMLState.ePMLState_EXECUTE AND fbPMLAuto.ePMLState <> Tc3_PackML.E_PMLState.ePMLState_STARTING, 	PT := T#30S);

tonConfectionEnding.Q;					tonConfectionEnding			(IN := (fbPMLAuto.ePMLState = Tc3_PackML.E_PMLState.ePMLState_COMPLETING OR fbPMLAuto.ePMLState = Tc3_PackML.E_PMLState.ePMLState_EXECUTE) AND VIS.bConfectionEnding AND tonEndOfConfecion.q);
tonTransporterStopping.Q;				tonTransporterStopping 		(IN := fbPMLAuto.ePMLState = Tc3_PackML.E_PMLState.ePMLState_STOPPING ,	 							PT := T#200MS);
tonDelayAfterReset.Q;					tonDelayAfterReset			(IN := GVL.bDelay40sAfterReset AND (fbPMLAuto.ePMLState = Tc3_PackML.E_PMLState.ePMLState_EXECUTE),	PT := tonLongDelayAfterStart.PT);//bylo 40S
tonDelayAfterBottleFeederDoorOpen.Q;	tonDelayAfterBottleFeederDoorOpen(IN:= GVL_IO.IbBottleFeederSafety, 															PT := T#3S);

rtLongDelayFirstDraging					(CLK := tonLongDelayFirstDraging.Q);
rtLongDelayFirstDragingLidFeeder		(CLK := tonLongDelayFirstDragingLidFeeder.Q);
rttonLongDelayAfterStart				(CLK := tonLongDelayAfterStart.Q);

fbbRecipeLoading						(bIN:=VIS.bRecipeLoading,	tFilterTimeOn:=T#0S,	tFilterTimeOff:=T#4S,	bOut=>); 
rtbRecipeLoading						(CLK :=VIS.bRecipeLoading);

//============================================================================


tonCheckFourthFormNotPresent		(IN:=NOT Main.IbFourthFormCheckFormSensor, PT:=T#100MS);
tonCheckFormSensorBetweenDispencer	(IN:= NOT Main.IbTwoPhasesFormSensorBetweenDispencers AND eBeforeDispencer12PackageState2Phase[1].bFormPresent
									 		AND eBeforeDispencer12PackageState2Phase[2].bFormPresent , PT:=T#150MS);
tonCheckFormBeforeDispencersGate	(IN:= NOT	MAIN.IbFourthFormCheckFormSensor AND NOT MAIN.IbFormCheckFormSensor AND 
											(P00_PackML.fbPMLAuto.ePMLState = E_PMLState.ePMLState_EXECUTE), PT:=T#5S); // dodana czasówka bo się rozjeżdzało przy rozpocząecoi konfekcji
MAIN.IbSecondFormCheckFormSensor;

IF tonDelayAfterReset.Q THEN
	GVL.bDelay40sAfterReset:=FALSE; //Kasuje bit po 40s, przeciąganie wraca do noramlnego trybu pracy i patrzy na ilośc formatek przed zakręcarkmi
END_IF;

//Licz for. przed doz. - do testów
tonIbFourthFormCheckFormSensor		(IN:=Main.IbFourthFormCheckFormSensor,	PT:=T#50MS);
rtIbFourthFormCheckFormSensor		(CLK:=tonIbFourthFormCheckFormSensor.Q,	Q=>);
IF rtIbFourthFormCheckFormSensor.Q THEN
	iFormsDragingFormCounter	:=	iFormsDragingFormCounter	+	1;
END_IF

//Do sprawdzenia, liczenie formatek
tofTransportersWorking(IN:= (P00_PackML.fbPMLAuto.ePMLState = E_PMLState.ePMLState_STARTING)	OR (P00_PackML.fbPMLAuto.ePMLState = E_PMLState.ePMLState_EXECUTE) OR 
							(P00_PackML.fbPMLAuto.ePMLState = E_PMLState.ePMLState_ABORTED) 	OR (P00_PackML.fbPMLAuto.ePMLState = E_PMLState.ePMLState_ABORTING) OR 
							(P00_PackML.fbPMLAuto.ePMLState = E_PMLState.ePMLState_STOPPING) 	OR (P00_PackML.fbPMLAuto.ePMLState = E_PMLState.ePMLState_STOPPED), PT:= T#3S);
tofTransportersWorking.Q;			   
rtResetAfterStart				(CLK:=tonLongDelayAfterStart.Q);
fbIbWeightFirstFormSensor		(bIn:=P05_Weight.IbWeight1FormSensor AND NOT bDosingTwoPhases,				tFilterTimeOn:=T#20MS, tFilterTimeOff:=T#20MS);//bylo 20MS
ftfbIbWeightFirstFormSensor		(CLK:=fbIbWeightFirstFormSensor.bOUT,					Q=>);

///////
fbIbWeightFirstForm2PhaseSensor(bIn:=P05_Weight.IbWeight5FormSensor AND bDosingTwoPhases, tFilterTimeon:=T#20MS, tFilterTimeOff:=T#20MS); // bylo 20Ms
ftfbIbWeightFirstForm2PhaseSensor(CLK:=fbIbWeightFirstForm2PhaseSensor.bOUT);

////
ACT_SignalsFormsCounting();
fbIbCapPuttedCheckFormSensor	(bIn:=P09_CapPuttedCheck.IbCapPuttedCheckFormSensor,	tFilterTimeOn:=T#20MS, tFilterTimeOff:=T#30MS); // bylo 20ms
fb2IbCapPuttedCheckFormSensor	(bIn:=P09_CapPuttedCheck.IbCapPuttedCheckFormSensor,	tFilterTimeOn:=T#3S, tFilterTimeOff:=T#20MS);//bylo 500ms
ftfbIbCapPuttedCheckFormSensor	(CLK:=fbIbCapPuttedCheckFormSensor.bOUT,				Q=>);

//Stacje są gotowe 
(*
bStationsAreReady := 
				(P01_BottleFeeder.fbBottleFeeder.eState = E_Station.eReady OR P01_BottleFeeder.fbBottleFeeder.eState = E_Station.eDisabled ) AND
				(P01_BottleFeeder.fbTurnTable.eState = E_Station.eReady OR P01_BottleFeeder.fbTurnTable.eState = E_Station.eDisabled) AND			
				(P01_PucksInserter.fbPucksInserter.eState = E_Station.eReady OR P01_PucksInserter.fbPucksInserter.eState = E_Station.eDisabled ) AND
				(P01_PucksInserter.fbTurnTable.eState = E_Station.eReady OR P01_PucksInserter.fbTurnTable.eState = E_Station.eDisabled) AND		
				(stBottleSorterRead.ePackMLAutoState = Tc3_PackML.E_PMLState.ePMLState_IDLE OR NOT stBottleSorterRead.bEnable OR bBottleSorterDisable) AND				
				(P02_Dispencers.fbDispencersDragRightStation.eState = E_Station.eReady OR P02_Dispencers.fbDispencersDragRightStation.eState = E_Station.eDisabled) AND 
				(P02_Dispencers.fbDispencersDragLeftStation.eState = E_Station.eReady OR P02_Dispencers.fbDispencersDragLeftStation.eState = E_Station.eDisabled) AND 
                (P02_Dispencers.fbDispencer1.eState = E_Station.eReady OR P02_Dispencers.fbDispencer1.eState = E_Station.eDisabled) AND
                (P02_Dispencers.fbDispencer2.eState = E_Station.eReady OR P02_Dispencers.fbDispencer2.eState = E_Station.eDisabled) AND
                (P02_Dispencers.fbDispencer3.eState = E_Station.eReady OR P02_Dispencers.fbDispencer3.eState = E_Station.eDisabled) AND
                (P02_Dispencers.fbDispencer4.eState = E_Station.eReady OR P02_Dispencers.fbDispencer4.eState = E_Station.eDisabled) AND
                (P02_Dispencers.fbDispencersCatch1Station.eState = E_Station.eReady OR  P02_Dispencers.fbDispencersCatch1Station.eState = E_Station.eDisabled) AND
                (P02_Dispencers.fbDispencersCatch2Station.eState = E_Station.eReady OR P02_Dispencers.fbDispencersCatch2Station.eState = E_Station.eDisabled) AND
                (P02_Dispencers.fbDispencersCatch3Station.eState = E_Station.eReady OR P02_Dispencers.fbDispencersCatch3Station.eState = E_Station.eDisabled) AND
                (P02_Dispencers.fbDispencersCatch4Station.eState = E_Station.eReady OR P02_Dispencers.fbDispencersCatch4Station.eState = E_Station.eDisabled) AND
				(P05_Weight.fbWeight1.eState  = E_Station.eReady OR P05_Weight.fbWeight1.eState = E_Station.eDisabled) AND
    			(P05_Weight.fbWeight2.eState  = E_Station.eReady OR P05_Weight.fbWeight2.eState = E_Station.eDisabled) AND
				(P05_Weight.fbWeight3.eState  = E_Station.eReady OR P05_Weight.fbWeight3.eState = E_Station.eDisabled) AND
				(P05_Weight.fbWeight4.eState  = E_Station.eReady OR P05_Weight.fbWeight4.eState = E_Station.eDisabled) AND
				(P05_Weight.fbWeight5.eState  = E_Station.eReady OR P05_Weight.fbWeight5.eState = E_Station.eDisabled) AND
				(P05_Weight.fbWeight6.eState  = E_Station.eReady OR P05_Weight.fbWeight6.eState = E_Station.eDisabled) AND				
				(P05_Weight.fbWeightStation.eState = E_Station.eReady OR P05_Weight.fbWeightStation.eState = E_Station.eDisabled) AND
				(P05_Weight.fbWeightStation2Phase.eState = E_Station.eReady OR P05_Weight.fbWeightStation2Phase.eState = E_Station.eDisabled) AND
				(P06_LidFeeder.fbLidFeeder.eState = E_Station.eReady OR P06_LidFeeder.fbLidFeeder.eState = E_Station.eDisabled) AND 
				(P06_LidFeeder.fbLidFeeder2.eState = E_Station.eReady OR P06_LidFeeder.fbLidFeeder2.eState = E_Station.eDisabled) AND
				(P06_LidFeeder.fbLidFeederDragStation.eState = E_Station.eReady OR P06_LidFeeder.fbLidFeederDragStation.eState = E_Station.eDisabled) AND
				//(P06_LidPuttedCheck.fbLidPuttedCheck.eState = E_Station.eReady OR P06_LidPuttedCheck.fbLidPuttedCheck.eState = E_Station.eDisabled) AND 
				(P06_LidSealer.fbLidSealer.eState = E_Station.eReady OR P06_LidSealer.fbLidSealer.eState = E_Station.eDisabled) AND 
				(P06_LidSealer.fbLidSealer2.eState = E_Station.eReady OR P06_LidSealer.fbLidSealer2.eState = E_Station.eDisabled) AND
				(P06_LidSealer.fbLidSealerDragStation.eState = E_Station.eReady OR P06_LidSealer.fbLidSealerDragStation.eState = E_Station.eDisabled) AND
				
				(P06_WickFeeder.fbWickFeederSt.eState = E_Station.eReady OR P06_WickFeeder.fbWickFeederSt.eState = E_Station.eDisabled) AND
				(P06_WickFeeder.fbWickFeederDragStation.eState = E_Station.eReady OR P06_WickFeeder.fbWickFeederDragStation.eState = E_Station.eDisabled) AND
				(P06_WickFeeder.fbWickFeederFormPositioning.eState = E_Station.eReady OR P06_WickFeeder.fbWickFeederFormPositioning.eState = E_Station.eDisabled) AND
				
				
				(P07_ROPP.fbROPPSlower.eState = E_Station.eReady  OR P07_ROPP.fbROPPSlower.eState = E_Station.eDisabled) AND
				(P07_ROPP.fbROPPFeeder.eState = E_Station.eReady  OR P07_ROPP.fbROPPFeeder.eState = E_Station.eDisabled) AND
				(P07_ROPP.fbROPPDrag.eState = E_Station.eReady  OR P07_ROPP.fbROPPDrag.eState = E_Station.eDisabled) AND
				(P07_ROPP.fbROPPCapping.eState = E_Station.eReady  OR P07_ROPP.fbROPPCapping.eState = E_Station.eDisabled) AND

				(P08_CapSorter.fbCapSorterDragStation.eState = E_Station.eReady OR P08_CapSorter.fbCapSorterDragStation.eState = E_Station.eDisabled) AND	
				(P08_CapFeeder.fbCapFeeder.eState = E_Station.eReady OR P08_CapFeeder.fbCapFeeder.eState = E_Station.eDisabled) AND
				(P08_CapSorter.fbCapSorterDragStation.eState = E_Station.eReady OR P08_CapSorter.fbCapSorterDragStation.eState = E_Station.eDisabled) AND
				(stCapSorterRead.ePackMLAutoState = Tc3_PackML.E_PMLState.ePMLState_IDLE OR NOT stCapSorterRead.bEnable OR bCapSorterDisable) AND 															
				(P09_CapPuttedCheck.fbCapPuttedCheck.eState = E_Station.eReady OR P09_CapPuttedCheck.fbCapPuttedCheck.eState = E_Station.eDisabled) AND
   				(P10_GripperScrewer.fbGripperScrewersDragStation.eState = E_Station.eReady  OR P10_GripperScrewer.fbGripperScrewersDragStation.eState = E_Station.eDisabled) AND
   	   			(P10_GripperScrewer.fbGripperScrewer1CatchStation.eState  = E_Station.eReady OR P10_GripperScrewer.fbGripperScrewer1CatchStation.eState = E_Station.eDisabled) AND
				(P10_GripperScrewer.fbGripperScrewer2CatchStation.eState  = E_Station.eReady OR P10_GripperScrewer.fbGripperScrewer2CatchStation.eState = E_Station.eDisabled) AND
    			(P11_CapCorrectCheck.fbCapCorrectCheck.eState = E_Station.eReady OR P11_CapCorrectCheck.fbCapCorrectCheck.eState = E_Station.eDisabled) AND
				(P13_BottleTransfer.fbBottleTransfer.eState = E_Station.eReady OR P13_BottleTransfer.fbBottleTransfer.eState = E_Station.eDisabled) AND 
				(P15_FormTransporters.fbFormTransporterDispencer.eState = E_Station.eReady OR P15_FormTransporters.fbFormTransporterDispencer.eState = E_Station.eDisabled) AND
				(P15_FormTransporters.fbFormTransporterScrewer.eState = E_Station.eReady OR P15_FormTransporters.fbFormTransporterScrewer.eState = E_Station.eDisabled) AND
 				(P15_FormTransporters.fbFormTransporterBeforeScrewer.eState = E_Station.eReady OR P15_FormTransporters.fbFormTransporterBeforeScrewer.eState = E_Station.eDisabled);		   
*)
// Czasówki od przeciągania dwufazowego
//Przejazd formatki
tonFourthFormat2PhaseSensor		(IN:= eBeforeDispencer34PackageState2Phase[2].bFormPresent AND MAIN.IbFourthFormCheckFormSensor AND (P00_PackML.fbPMLAuto.ePMLState = E_PMLState.ePMLState_EXECUTE));
tonSecondForm2PhaseSensor		(IN:= Main.IbTwoPhasesFormSensorBetweenDispencers AND eBeforeDispencer12PackageState2Phase[1].bFormPresent AND eBeforeDispencer12PackageState2Phase[2].bFormPresent AND (P00_PackML.fbPMLAuto.ePMLState = E_PMLState.ePMLState_EXECUTE), PT:=T#600MS);

// Czasówka dodana na potrzeby zadziałania naprawy jak coś zle przesunie 02.06 Damian
tonSecondForm2PhaseSensorRepair(IN:=Main.IbTwoPhasesFormSensorBetweenDispencers AND NOT eBeforeDispencer12PackageState2Phase[1].bFormPresent AND (P00_PackML.fbPMLAuto.ePMLState = E_PMLState.ePMLState_EXECUTE), PT:=T#15S);

// Czasowka zamiast P10_GripperScrewer.IbDragMiddleSensor 
tonGripperScrewerDragMiddleSensor	(IN:=P10_GripperScrewer.fbGripperScrewersDragStation.eRunningState >= E_DragStationState.eDraging, PT:=T#300MS);

// Czasowka zamiast Ppozycji przeciągania pod dozownikami
tonDispencersDragLeftMiddleSensor	(IN:=P02_Dispencers.fbDispencersDragLeftStation.eRunningState >= E_DragStationState.eDraging, PT:=T#200MS);
tonDispencersDragRightMiddleSensor	(IN:=P02_Dispencers.fbDispencersDragRightStation.eRunningState >= E_DragStationState.eDraging, PT:=T#200MS);

// Czasowka zamiast pozycji przeciągania pod sorterem nasadek
tonCapSorterDragMiddleSensor		(IN:=P08_CapSorter.fbCapSorterDragStation.eRunningState >= E_DragStationState.eDraging, PT:=T#200MS);
tonIbCapSorterAfterFormSensor		(IN:=NOT MAIN.IbCapSorterAfterFormSensor AND NOT MAIN.IbCapSorterAfterFormSensor2, PT:=T#100MS);//bylo 300
tonIbCapSorterAfterFormSensor3		(IN:=MAIN.IbCapSorterAfterFormSensor3, PT:=T#2S);//bylo 500

tonbCapSorterOrCapSorterDragError 	(IN:=fbPMLAuto.ePMLState = Tc3_PackML.E_PMLState.ePMLState_STOPPING AND stCapSorterRead.eError.bError OR P08_CapSorter.fbCapSorterDragStation.eState = E_Station.eError OR GeneralAlarms.nErrorCode=38, PT:=T#7S);

//Czasówka do przy przełączaniu 2 fazy 
fbIbFourthFormCheckFormSensor				(bIn:=MAIN.IbFourthFormCheckFormSensor, 			tFilterTimeOn:=T#2S, tFilterTimeOff:=T#2S);
fbIbTwoPhasesFormSensorBetweenDispencers 	(bIn:=Main.IbTwoPhasesFormSensorBetweenDispencers,	tFilterTimeOn:=T#500MS, tFilterTimeOff:=T#2S);
fbIbSecondFormCheckFormSensor				(bIn:=MAIN.IbSecondFormCheckFormSensor,				tFilterTimeOn:=T#2S, tFilterTimeOff:=T#2S);
tofbDosingTwoPhases							(IN:=bDosingTwoPhases,	PT:=T#20S);
// Czasówki od przeciągania 1 faza

// czasówki uzaleźnione od prędkości transportera
IF bChangeOver THEN
	tonFourthFormatSensor.PT:=T#5S;
ELSIF GVL.nFormTransportersDispencerVelocitySV <1000 AND NOT brtLongDelayFirstDraging THEN
	tonFourthFormatSensor.PT:=T#800MS;//bylo 400 dp	
ELSIF  (GVL.nFormTransportersDispencerVelocitySV >=1000 AND GVL.nFormTransportersDispencerVelocitySV <1300) AND NOT brtLongDelayFirstDraging THEN
	tonFourthFormatSensor.PT:=T#700MS; //bylo 500 //350 się nie sprawdza
ELSIF (GVL.nFormTransportersDispencerVelocitySV >=1300) AND NOT brtLongDelayFirstDraging THEN
	tonFourthFormatSensor.PT:=T#600MS; //bylo 300
ELSIF brtLongDelayFirstDraging THEN
	tonFourthFormatSensor.PT:=T#1000MS;
END_IF
//Przejazd formatki
tonFourthFormatSensor			(IN:= eBeforeDispencersPackageState[4].bFormPresent AND MAIN.IbFourthFormCheckFormSensor AND MAIN.IbSecondFormCheckFormSensor AND (P00_PackML.fbPMLAuto.ePMLState = E_PMLState.ePMLState_EXECUTE));
tonFourthFormatSensor2			(IN:= eBeforeDispencersPackageState[4].bFormPresent AND MAIN.IbFourthFormCheckFormSensor AND MAIN.IbSecondFormCheckFormSensor AND (P00_PackML.fbPMLAuto.ePMLState = E_PMLState.ePMLState_EXECUTE) AND bCapSorterDragIfNot4PucksAnd5sRepair, PT:=T#2S);


// czasówki uzaleźnione od prędkości transportera
IF GVL.nFormTransportersScrewerVelocitySV <1000 AND NOT brtLongDelayFirstDraging THEN
	tonCapSorterFourthFormatSensorAnRegister.PT:=T#100MS;	 	
ELSIF  (GVL.nFormTransportersScrewerVelocitySV >=1000 AND GVL.nFormTransportersScrewerVelocitySV <1300) AND NOT brtLongDelayFirstDraging THEN
	tonCapSorterFourthFormatSensorAnRegister.PT:=T#100MS;		
ELSIF (GVL.nFormTransportersScrewerVelocitySV >=1300) AND NOT brtLongDelayFirstDraging THEN
	tonCapSorterFourthFormatSensorAnRegister.PT:=T#100MS;	
ELSIF brtLongDelayFirstDraging THEN
	tonCapSorterFourthFormatSensorAnRegister.PT:=T#1000MS;
END_IF
tonCapSorterFourthFormatSensorAnRegister			(IN:=	eBeforeCapSorterPackageState[4].bFormPresent	AND fbIbCapSorterFourthFormCheckFormSensor.bOut AND (P00_PackML.fbPMLAuto.ePMLState = E_PMLState.ePMLState_EXECUTE OR P00_PackML.fbPMLAuto.ePMLState = E_PMLState.ePMLState_STOPPING));
tonIbCapSorterFirstFormCheckFormSensor				(IN:=	MAIN.IbCapSorterFirstFormCheckFormSensor,PT:=T#30MS);
fbIbCapSorterFourthFormCheckFormSensor				(bIN:= MAIN.IbCapSorterFourthFormCheckFormSensor, tFilterTimeOn:=T#40MS, tFilterTimeOff:=T#40MS, bOut=>);
IF VIS.nFormTransportersScrewerVelocitySVShow < 500 THEN
	tonCapSorterFourthFormatSensor		(IN:=	fbIbCapSorterFourthFormCheckFormSensor.bOut 		, PT:=T#200MS);
ELSE
	tonCapSorterFourthFormatSensor		(IN:=	fbIbCapSorterFourthFormCheckFormSensor.bOut 		, PT:=T#40MS);
END_IF
tonCapSorterFourthFormatSensorStarting		(IN:=	tonCapSorterFourthFormatSensor.Q					, PT:=T#1S);
tonbFormTransportersAfterCapSorterCmdStart	(IN:=	bFormTransportersAfterCapSorterCmdStart				, PT:=T#1S);
rttonCapSorterFourthFormatSensorCounter	(CLK:=	tonCapSorterFourthFormatSensor.Q			,Q=>);			
IF rttonCapSorterFourthFormatSensorCounter.Q THEN
	iCapSorterDragFormCounter := iCapSorterDragFormCounter	+	1;
END_IF

tonLidSealerSecondFormatSensor (IN:= (*	eBeforeLidSealerPackageState[2].bFormPresent AND *) MAIN.IbLidSealerSecondFormSensor AND 
								(P00_PackML.fbPMLAuto.ePMLState = E_PMLState.ePMLState_EXECUTE OR P00_PackML.fbPMLAuto.ePMLState = E_PMLState.ePMLState_STOPPING),
								PT:=T#200MS);

rttonLidSealerSecondFormatSensorCounter (CLK:= tonLidSealerSecondFormatSensor.Q);
IF rttonLidSealerSecondFormatSensorCounter.Q THEN
	 iLidSealerDragFormCounter := iLidSealerDragFormCounter + 1;
END_IF


toffbDispencersDragLeftStationbCycleDone.ET;
toffbDispencersDragLeftStationbCycleDone.Q;
toffbDispencersDragLeftStationbCycleDone(IN:=P02_Dispencers.fbDispencersDragLeftStation.eRunningState = E_DragStationState.eDraging, PT:=T#3S);
		
//Na conajmniej jednej ze stacji włączono bazowanie
bHomingIsOnAtLeastOneStation 		:= 
									VIS.bBottleFeederHoming	OR		
									VIS.bPucksInserterHoming OR		
									(stBottleSorterWrite.bHoming OR stBottleSorterRead.bHoming) OR		
									VIS.bDispencersHoming OR     
									VIS.bFormsDragingRightHoming OR	
									VIS.bFormsDragingLeftHoming OR
									VIS.bWeightLiftHoming OR			
									VIS.bCapFeederHoming OR	
									VIS.bWickFeederHoming OR	
									VIS.bWickFeederDragingHoming OR			
									VIS.bLidFeederHoming OR	
									VIS.bLidFeederDragingHoming OR	
									Vis.bWickFeederDragingHoming OR
									Vis.bWickFeederHoming OR	
									//VIS.bLidPuttedCheckHoming OR	
									VIS.bLidSealerHoming OR		
									VIS.bLidSealerDragingHoming OR		
									VIS_ROPP.bROPPFeederHoming OR	
									VIS_ROPP.bROPPDragHoming OR	
									VIS_ROPP.bROPPCappingHoming OR	
									VIS.bCapSorterDragHoming OR		
									(stCapSorterWrite.bHoming OR stCapSorterRead.bHoming) OR 			
									VIS.bCapPuttedCheckHoming OR		
									VIS.bGripperScrewerHoming OR		
									VIS.bBottleDragingStationHoming OR	
									VIS.bCapCorrectCheckHoming OR      
									VIS.bBottleTransferHoming
									; 																	
									
//Jedna ze stacji wymaga bazowania
bAtLeastOneOfTheStationsNeedHoming 	:= 
									(NOT P01_BottleFeeder.fbBottleFeeder.bHomingDone AND P01_BottleFeeder.fbBottleFeeder.bEnable) OR
									(NOT P01_PucksInserter.fbPucksInserter.bHomingDone AND P01_PucksInserter.fbPucksInserter.bEnable) OR									
									(NOT stBottleSorterRead.bHomingDone AND stBottleSorterRead.bEnable AND NOT bBottleSorterDisable) OR
									(NOT P02_Dispencers.fbDispencersDragRightStation.bHomingDone AND GVL.bFormsDragingRightEnable) OR
									(NOT P02_Dispencers.fbDispencersDragLeftStation.bHomingDone AND GVL.bFormsDragingLeftEnable) OR
									(NOT P02_Dispencers.fbDispencer1.bHomingDone AND bDispencer1Enable) OR
									(NOT P02_Dispencers.fbDispencer2.bHomingDone AND bDispencer2Enable) OR
									(NOT P02_Dispencers.fbDispencer3.bHomingDone AND bDispencer3Enable) OR
									(NOT P02_Dispencers.fbDispencer4.bHomingDone AND bDispencer4Enable) OR
									(NOT P02_Dispencers.fbDispencersCatch1Station.bHomingDone AND 
									 NOT P02_Dispencers.fbDispencersCatch2Station.bHomingDone AND
									 NOT P02_Dispencers.fbDispencersCatch3Station.bHomingDone AND 
									 NOT P02_Dispencers.fbDispencersCatch4Station.bHomingDone AND
									(bDispencer1Enable OR bDispencer2Enable OR bDispencer3Enable OR bDispencer4Enable)) OR
									(NOT P05_Weight.fbWeightStation.bHomingDone AND bWeightLiftEnable) OR
									(NOT P05_Weight.fbWeightStation2Phase.bHomingDone AND bWeightLiftEnable AND bDosingTwoPhases) OR
									(NOT P06_LidFeeder.fbLidFeeder.bHomingDone AND bLidFeederEnable) OR
									(NOT P06_LidFeeder.fbLidFeeder2.bHomingDone AND bLidFeederEnable) OR 
									(NOT P06_LidFeeder.fbLidFeederDragStation.bHomingDone AND bLidFeederDragingStationEnable) OR								
									//(NOT P06_LidPuttedCheck.fbLidPuttedCheck.bHomingDone AND bLidPuttedCheckEnable) OR
									(NOT P06_LidSealer.fbLidSealer.bHomingDone AND bLidSealerEnable) OR
									(NOT P06_LidSealer.fbLidSealer2.bHomingDone AND bLidSealerEnable) OR
									(NOT P06_LidSealer.fbLidSealerDragStation.bHomingDone AND bLidSealerDragingStationEnable) OR

									(NOT P06_WickFeeder.fbWickFeederSt.bHomingDone AND bWickFeederEnable) OR
									(NOT P06_WickFeeder.fbWickFeederDragStation.bHomingDone AND bWickFeederDragingStationEnable) OR

									(NOT P07_ROPP.fbROPPFeeder.bHomingDone AND bROPPFeederEnable) OR
									(NOT P07_ROPP.fbROPPDrag.bHomingDone AND bROPPDragEnable) OR
									(NOT P07_ROPP.fbROPPCapping.bHomingDone AND bROPPCappingEnable) OR

									(NOT P08_CapFeeder.fbCapFeeder.bHomingDone AND bCapFeederEnable) OR 
									(NOT P08_CapSorter.fbCapSorterDragStation.bHomingDone AND bCapSorterDragEnable) OR
									(NOT stCapSorterRead.bHomingDone AND stCapSorterRead.bEnable AND NOT bCapSorterDisable) OR
									(NOT P09_CapPuttedCheck.fbCapPuttedCheck.bHomingDone AND bCapPuttedCheckEnable) OR
									(NOT P10_GripperScrewer.fbGripperScrewersDragStation.bHomingDone AND bBottleDragingStationEnable) OR
									(NOT P10_GripperScrewer.fb2GripperScrewer1.bHomingDone AND bGripperScrewer1Enable) OR
									(NOT P10_GripperScrewer.fb2GripperScrewer2.bHomingDone AND bGripperScrewer2Enable) OR	
									(NOT P10_GripperScrewer.fbGripperScrewer1CatchStation.bHomingDone AND bGripperScrewer1Enable) OR
									(NOT P10_GripperScrewer.fbGripperScrewer2CatchStation.bHomingDone AND bGripperScrewer2Enable) OR
									(NOT P10_GripperScrewer.fbGripperScrewersDragStation.bHomingDone AND bBottleDragingStationEnable) OR
									(NOT P11_CapCorrectCheck.fbCapCorrectCheck.bHomingDone AND bCapCorrectCheckEnable) OR
									(NOT P13_BottleTransfer.fbBottleTransfer.bHomingDone AND P13_BottleTransfer.fbBottleTransfer.bEnable) 
									;

//Stacje są gotowe
bStationsAreReady :=  
				(P01_BottleFeeder.fbBottleFeeder.eState = E_Station.eReady OR P01_BottleFeeder.fbBottleFeeder.eState = E_Station.eDisabled ) AND
				(P01_BottleFeeder.fbTurnTable.eState = E_Station.eReady OR P01_BottleFeeder.fbTurnTable.eState = E_Station.eDisabled) AND
				(P01_PucksInserter.fbPucksInserter.eState = E_Station.eReady OR P01_PucksInserter.fbPucksInserter.eState = E_Station.eDisabled ) AND
				//(P01_PucksInserter.fbTurnTable.eState = E_Station.eReady OR P01_PucksInserter.fbTurnTable.eState = E_Station.eDisabled) AND
				((stBottleSorterRead.ePackMLAutoState = Tc3_PackML.E_PMLState.ePMLState_IDLE OR NOT stBottleSorterRead.bEnable OR bBottleSorterDisable) ) AND
				(P02_Dispencers.fbDispencersDragRightStation.eState = E_Station.eReady OR P02_Dispencers.fbDispencersDragRightStation.eState = E_Station.eDisabled) AND 
				(P02_Dispencers.fbDispencersDragLeftStation.eState = E_Station.eReady OR P02_Dispencers.fbDispencersDragLeftStation.eState = E_Station.eDisabled) AND 
                (P02_Dispencers.fbDispencer1.eState = E_Station.eReady OR P02_Dispencers.fbDispencer1.eState = E_Station.eDisabled) AND
                (P02_Dispencers.fbDispencer2.eState = E_Station.eReady OR P02_Dispencers.fbDispencer2.eState = E_Station.eDisabled) AND
                (P02_Dispencers.fbDispencer3.eState = E_Station.eReady OR P02_Dispencers.fbDispencer3.eState = E_Station.eDisabled) AND
                (P02_Dispencers.fbDispencer4.eState = E_Station.eReady OR P02_Dispencers.fbDispencer4.eState = E_Station.eDisabled) AND
                (P02_Dispencers.fbDispencersCatch1Station.eState = E_Station.eReady OR  P02_Dispencers.fbDispencersCatch1Station.eState = E_Station.eDisabled) AND
                (P02_Dispencers.fbDispencersCatch2Station.eState = E_Station.eReady OR P02_Dispencers.fbDispencersCatch2Station.eState = E_Station.eDisabled) AND
                (P02_Dispencers.fbDispencersCatch3Station.eState = E_Station.eReady OR P02_Dispencers.fbDispencersCatch3Station.eState = E_Station.eDisabled) AND
                (P02_Dispencers.fbDispencersCatch4Station.eState = E_Station.eReady OR P02_Dispencers.fbDispencersCatch4Station.eState = E_Station.eDisabled) AND
				(P05_Weight.fbWeight1.eState  = E_Station.eReady OR P05_Weight.fbWeight1.eState = E_Station.eDisabled) AND
    			(P05_Weight.fbWeight2.eState  = E_Station.eReady OR P05_Weight.fbWeight2.eState = E_Station.eDisabled) AND
				(P05_Weight.fbWeight3.eState  = E_Station.eReady OR P05_Weight.fbWeight3.eState = E_Station.eDisabled) AND
				(P05_Weight.fbWeight4.eState  = E_Station.eReady OR P05_Weight.fbWeight4.eState = E_Station.eDisabled) AND
				(P05_Weight.fbWeight5.eState  = E_Station.eReady OR P05_Weight.fbWeight5.eState = E_Station.eDisabled) AND
				(P05_Weight.fbWeight6.eState  = E_Station.eReady OR P05_Weight.fbWeight6.eState = E_Station.eDisabled) AND				
				(P05_Weight.fbWeightStation.eState = E_Station.eReady OR P05_Weight.fbWeightStation.eState = E_Station.eDisabled) AND
				(P05_Weight.fbWeightStation2Phase.eState = E_Station.eReady OR P05_Weight.fbWeightStation2Phase.eState = E_Station.eDisabled) AND
				(P06_LidFeeder.fbLidFeeder.eState = E_Station.eReady OR P06_LidFeeder.fbLidFeeder.eState = E_Station.eDisabled) AND 
				(P06_LidFeeder.fbLidFeeder2.eState = E_Station.eReady OR P06_LidFeeder.fbLidFeeder2.eState = E_Station.eDisabled) AND
				(P06_LidFeeder.fbLidFeederDragStation.eState = E_Station.eReady OR P06_LidFeeder.fbLidFeederDragStation.eState = E_Station.eDisabled) AND
				//(P06_LidPuttedCheck.fbLidPuttedCheck.eState = E_Station.eReady OR P06_LidPuttedCheck.fbLidPuttedCheck.eState = E_Station.eDisabled) AND 
				(P06_LidSealer.fbLidSealer.eState = E_Station.eReady OR P06_LidSealer.fbLidSealer.eState = E_Station.eDisabled) AND 
				(P06_LidSealer.fbLidSealer2.eState = E_Station.eReady OR P06_LidSealer.fbLidSealer2.eState = E_Station.eDisabled) AND
				(P06_LidSealer.fbLidSealerDragStation.eState = E_Station.eReady OR P06_LidSealer.fbLidSealerDragStation.eState = E_Station.eDisabled) AND
				
				(P06_WickFeeder.fbWickFeederSt.eState = E_Station.eReady OR P06_WickFeeder.fbWickFeederSt.eState = E_Station.eDisabled) AND
				(P06_WickFeeder.fbWickFeederDragStation.eState = E_Station.eReady OR P06_WickFeeder.fbWickFeederDragStation.eState = E_Station.eDisabled) AND

				(P07_ROPP.fbROPPFeeder.eState = E_Station.eReady OR P07_ROPP.fbROPPFeeder.eState = E_Station.eDisabled) AND
				(P07_ROPP.fbROPPDrag.eState = E_Station.eReady OR P07_ROPP.fbROPPDrag.eState = E_Station.eDisabled) AND
				(P07_ROPP.fbROPPCapping.eState = E_Station.eReady OR P07_ROPP.fbROPPCapping.eState = E_Station.eDisabled) AND

				(P08_CapFeeder.fbCapFeeder.eState = E_Station.eReady OR P08_CapFeeder.fbCapFeeder.eState = E_Station.eDisabled) AND
				(P08_CapSorter.fbCapSorterDragStation.eState = E_Station.eReady OR P08_CapSorter.fbCapSorterDragStation.eState = E_Station.eDisabled) AND				
				((stCapSorterRead.ePackMLAutoState = Tc3_PackML.E_PMLState.ePMLState_IDLE OR NOT stCapSorterRead.bEnable OR bCapSorterDisable) ) AND 				
				(P09_CapPuttedCheck.fbCapPuttedCheck.eState = E_Station.eReady OR P09_CapPuttedCheck.fbCapPuttedCheck.eState = E_Station.eDisabled) AND
   				(P10_GripperScrewer.fbGripperScrewersDragStation.eState = E_Station.eReady  OR P10_GripperScrewer.fbGripperScrewersDragStation.eState = E_Station.eDisabled) AND
   	   			(P10_GripperScrewer.fbGripperScrewer1CatchStation.eState  = E_Station.eReady OR P10_GripperScrewer.fbGripperScrewer1CatchStation.eState = E_Station.eDisabled) AND
				(P10_GripperScrewer.fbGripperScrewer2CatchStation.eState  = E_Station.eReady OR P10_GripperScrewer.fbGripperScrewer2CatchStation.eState = E_Station.eDisabled) AND
    			(P11_CapCorrectCheck.fbCapCorrectCheck.eState  = E_Station.eReady OR P11_CapCorrectCheck.fbCapCorrectCheck.eState = E_Station.eDisabled) AND
				(P13_BottleTransfer.fbBottleTransfer.eState = E_Station.eReady OR P13_BottleTransfer.fbBottleTransfer.eState = E_Station.eDisabled) AND 
				(P15_FormTransporters.fbFormTransporterDispencer.eState = E_Station.eReady OR P15_FormTransporters.fbFormTransporterDispencer.eState = E_Station.eDisabled) AND
				(P15_FormTransporters.fbFormTransporterScrewer.eState = E_Station.eReady OR P15_FormTransporters.fbFormTransporterScrewer.eState = E_Station.eDisabled) AND
				(P15_FormTransporters.fbFormTransporterROPP.eState = E_Station.eReady OR P15_FormTransporters.fbFormTransporterROPP.eState = E_Station.eDisabled) AND
 				(P15_FormTransporters.fbFormTransporterBeforeScrewer.eState = E_Station.eReady OR P15_FormTransporters.fbFormTransporterBeforeScrewer.eState = E_Station.eDisabled)
				;	
									   					
//Stacje są gotowe albo w manualu 
bStationsAreReadyOrManual := 
				(P01_BottleFeeder.fbBottleFeeder.eState = E_Station.eReady OR P01_BottleFeeder.fbBottleFeeder.eState = E_Station.eManualMovement OR P01_BottleFeeder.fbBottleFeeder.eState = E_Station.eDisabled ) AND
				(P01_BottleFeeder.fbTurnTable.eState = E_Station.eReady OR P01_BottleFeeder.fbTurnTable.eState = E_Station.eManualMovement OR P01_BottleFeeder.fbTurnTable.eState = E_Station.eDisabled) AND
				(P01_PucksInserter.fbPucksInserter.eState = E_Station.eReady OR P01_PucksInserter.fbPucksInserter.eState = E_Station.eManualMovement OR P01_PucksInserter.fbPucksInserter.eState = E_Station.eDisabled) AND
				//(P01_PucksInserter.fbTurnTable.eState = E_Station.eReady OR P01_PucksInserter.fbTurnTable.eState = E_Station.eManualMovement OR P01_PucksInserter.fbTurnTable.eState = E_Station.eDisabled) AND
				(stBottleSorterRead.ePackMLAutoState = E_PMLState.ePMLState_RESETTING OR stBottleSorterRead.ePackMLAutoState = E_PMLState.ePMLState_IDLE OR NOT stBottleSorterRead.bEnable OR bBottleSorterDisable)  AND
				(P02_Dispencers.fbDispencersDragRightStation.eState = E_Station.eReady OR P02_Dispencers.fbDispencersDragRightStation.eState = E_Station.eManualMovement OR P02_Dispencers.fbDispencersDragRightStation.eState = E_Station.eDisabled) AND 
				(P02_Dispencers.fbDispencersDragLeftStation.eState = E_Station.eReady OR P02_Dispencers.fbDispencersDragLeftStation.eState = E_Station.eManualMovement OR P02_Dispencers.fbDispencersDragLeftStation.eState = E_Station.eDisabled) AND 
                (P02_Dispencers.fbDispencer1.eState = E_Station.eReady OR P02_Dispencers.fbDispencer1.eState = E_Station.eManualMovement OR P02_Dispencers.fbDispencer1.eState = E_Station.eDisabled) AND
                (P02_Dispencers.fbDispencer2.eState = E_Station.eReady OR P02_Dispencers.fbDispencer2.eState = E_Station.eManualMovement OR P02_Dispencers.fbDispencer2.eState = E_Station.eDisabled) AND
                (P02_Dispencers.fbDispencer3.eState = E_Station.eReady OR P02_Dispencers.fbDispencer3.eState = E_Station.eManualMovement OR P02_Dispencers.fbDispencer3.eState = E_Station.eDisabled) AND
                (P02_Dispencers.fbDispencer4.eState = E_Station.eReady OR P02_Dispencers.fbDispencer4.eState = E_Station.eManualMovement OR P02_Dispencers.fbDispencer4.eState = E_Station.eDisabled) AND
                (P02_Dispencers.fbDispencersCatch1Station.eState = E_Station.eReady OR P02_Dispencers.fbDispencersCatch1Station.eState = E_Station.eManualMovement OR P02_Dispencers.fbDispencersCatch1Station.eState = E_Station.eDisabled) AND
                (P02_Dispencers.fbDispencersCatch2Station.eState = E_Station.eReady OR P02_Dispencers.fbDispencersCatch2Station.eState = E_Station.eManualMovement OR P02_Dispencers.fbDispencersCatch2Station.eState = E_Station.eDisabled) AND
                (P02_Dispencers.fbDispencersCatch3Station.eState = E_Station.eReady OR P02_Dispencers.fbDispencersCatch3Station.eState = E_Station.eManualMovement OR P02_Dispencers.fbDispencersCatch3Station.eState = E_Station.eDisabled) AND
                (P02_Dispencers.fbDispencersCatch4Station.eState = E_Station.eReady OR P02_Dispencers.fbDispencersCatch4Station.eState = E_Station.eManualMovement OR P02_Dispencers.fbDispencersCatch4Station.eState = E_Station.eDisabled) AND
				(P05_Weight.fbWeight1.eState = E_Station.eReady OR P05_Weight.fbWeight1.eState = E_Station.eManualMovement OR P05_Weight.fbWeight1.eState = E_Station.eDisabled) AND
    			(P05_Weight.fbWeight2.eState = E_Station.eReady OR P05_Weight.fbWeight2.eState = E_Station.eManualMovement OR P05_Weight.fbWeight2.eState = E_Station.eDisabled) AND
				(P05_Weight.fbWeight3.eState = E_Station.eReady OR P05_Weight.fbWeight3.eState = E_Station.eManualMovement OR P05_Weight.fbWeight3.eState = E_Station.eDisabled) AND
				(P05_Weight.fbWeight4.eState = E_Station.eReady OR P05_Weight.fbWeight4.eState = E_Station.eManualMovement OR P05_Weight.fbWeight4.eState = E_Station.eDisabled) AND
				(P05_Weight.fbWeight5.eState = E_Station.eReady OR P05_Weight.fbWeight5.eState = E_Station.eManualMovement OR P05_Weight.fbWeight5.eState = E_Station.eDisabled) AND
				(P05_Weight.fbWeight6.eState = E_Station.eReady OR P05_Weight.fbWeight6.eState = E_Station.eManualMovement OR P05_Weight.fbWeight6.eState = E_Station.eDisabled) AND				
				(P05_Weight.fbWeightStation.eState = E_Station.eReady OR P05_Weight.fbWeightStation.eState = E_Station.eManualMovement OR P05_Weight.fbWeightStation.eState = E_Station.eDisabled) AND
				(P05_Weight.fbWeightStation2Phase.eState = E_Station.eReady OR P05_Weight.fbWeightStation2Phase.eState = E_Station.eManualMovement OR P05_Weight.fbWeightStation2Phase.eState = E_Station.eDisabled) AND
				(P06_LidFeeder.fbLidFeeder.eState = E_Station.eReady OR P06_LidFeeder.fbLidFeeder.eState = E_Station.eManualMovement OR P06_LidFeeder.fbLidFeeder.eState = E_Station.eDisabled) AND 
				(P06_LidFeeder.fbLidFeeder2.eState = E_Station.eReady OR P06_LidFeeder.fbLidFeeder2.eState = E_Station.eManualMovement OR P06_LidFeeder.fbLidFeeder2.eState = E_Station.eDisabled) AND
				(P06_LidFeeder.fbLidFeederDragStation.eState = E_Station.eReady OR P06_LidFeeder.fbLidFeederDragStation.eState = E_Station.eManualMovement OR P06_LidFeeder.fbLidFeederDragStation.eState = E_Station.eDisabled) AND
				//(P06_LidPuttedCheck.fbLidPuttedCheck.eState = E_Station.eReady OR P06_LidPuttedCheck.fbLidPuttedCheck.eState = E_Station.eManualMovement OR P06_LidPuttedCheck.fbLidPuttedCheck.eState = E_Station.eDisabled) AND 
				(P06_LidSealer.fbLidSealer.eState = E_Station.eReady OR P06_LidSealer.fbLidSealer.eState = E_Station.eManualMovement OR P06_LidSealer.fbLidSealer.eState = E_Station.eDisabled) AND 
				(P06_LidSealer.fbLidSealer2.eState = E_Station.eReady OR P06_LidSealer.fbLidSealer2.eState = E_Station.eManualMovement OR P06_LidSealer.fbLidSealer2.eState = E_Station.eDisabled) AND
				(P06_LidSealer.fbLidSealerDragStation.eState = E_Station.eReady OR P06_LidSealer.fbLidSealerDragStation.eState = E_Station.eManualMovement OR P06_LidSealer.fbLidSealerDragStation.eState = E_Station.eDisabled) AND
				
				(P06_WickFeeder.fbWickFeederSt.eState = E_Station.eReady OR P06_WickFeeder.fbWickFeederSt.eState = E_Station.eManualMovement OR P06_WickFeeder.fbWickFeederSt.eState = E_Station.eDisabled) AND
				(P06_WickFeeder.fbWickFeederDragStation.eState = E_Station.eReady OR P06_WickFeeder.fbWickFeederDragStation.eState = E_Station.eManualMovement OR P06_WickFeeder.fbWickFeederDragStation.eState = E_Station.eDisabled) AND
				
			
				(P07_ROPP.fbROPPFeeder.eState = E_Station.eReady OR P07_ROPP.fbROPPFeeder.eState = E_Station.eManualMovement OR P07_ROPP.fbROPPFeeder.eState = E_Station.eDisabled) AND
				(P07_ROPP.fbROPPDrag.eState = E_Station.eReady OR P07_ROPP.fbROPPDrag.eState = E_Station.eManualMovement OR P07_ROPP.fbROPPDrag.eState = E_Station.eDisabled) AND
				(P07_ROPP.fbROPPCapping.eState = E_Station.eReady OR P07_ROPP.fbROPPCapping.eState = E_Station.eManualMovement OR P07_ROPP.fbROPPCapping.eState = E_Station.eDisabled) AND

				(P08_CapFeeder.fbCapFeeder.eState = E_Station.eReady OR P08_CapFeeder.fbCapFeeder.eState = E_Station.eManualMovement OR P08_CapFeeder.fbCapFeeder.eState = E_Station.eDisabled) AND
				(P08_CapSorter.fbCapSorterDragStation.eState = E_Station.eReady OR P08_CapSorter.fbCapSorterDragStation.eState = E_Station.eManualMovement OR P08_CapSorter.fbCapSorterDragStation.eState = E_Station.eDisabled) AND				
				(stCapSorterRead.ePackMLAutoState = E_PMLState.ePMLState_RESETTING OR stCapSorterRead.ePackMLAutoState = E_PMLState.ePMLState_IDLE OR NOT stCapSorterRead.bEnable OR bCapSorterDisable)  AND				
				(P09_CapPuttedCheck.fbCapPuttedCheck.eState = E_Station.eReady OR P09_CapPuttedCheck.fbCapPuttedCheck.eState = E_Station.eManualMovement OR P09_CapPuttedCheck.fbCapPuttedCheck.eState = E_Station.eDisabled) AND
   				(P10_GripperScrewer.fbGripperScrewersDragStation.eState = E_Station.eReady OR P10_GripperScrewer.fbGripperScrewersDragStation.eState = E_Station.eManualMovement OR P10_GripperScrewer.fbGripperScrewersDragStation.eState = E_Station.eDisabled) AND
   	   			(P10_GripperScrewer.fbGripperScrewer1CatchStation.eState = E_Station.eReady OR P10_GripperScrewer.fbGripperScrewer1CatchStation.eState = E_Station.eManualMovement OR P10_GripperScrewer.fbGripperScrewer1CatchStation.eState = E_Station.eDisabled) AND
				(P10_GripperScrewer.fbGripperScrewer2CatchStation.eState = E_Station.eReady OR P10_GripperScrewer.fbGripperScrewer2CatchStation.eState = E_Station.eManualMovement OR P10_GripperScrewer.fbGripperScrewer2CatchStation.eState = E_Station.eDisabled) AND
    			(P11_CapCorrectCheck.fbCapCorrectCheck.eState = E_Station.eReady OR P11_CapCorrectCheck.fbCapCorrectCheck.eState = E_Station.eManualMovement OR P11_CapCorrectCheck.fbCapCorrectCheck.eState = E_Station.eDisabled) AND
				(P13_BottleTransfer.fbBottleTransfer.eState = E_Station.eReady OR P13_BottleTransfer.fbBottleTransfer.eState = E_Station.eManualMovement OR P13_BottleTransfer.fbBottleTransfer.eState = E_Station.eDisabled) AND 
				(P15_FormTransporters.fbFormTransporterDispencer.eState = E_Station.eReady OR P15_FormTransporters.fbFormTransporterDispencer.eState = E_Station.eManualMovement OR P15_FormTransporters.fbFormTransporterDispencer.eState = E_Station.eDisabled) AND
				(P15_FormTransporters.fbFormTransporterScrewer.eState = E_Station.eReady OR P15_FormTransporters.fbFormTransporterScrewer.eState = E_Station.eManualMovement OR P15_FormTransporters.fbFormTransporterScrewer.eState = E_Station.eDisabled) AND
 				(P15_FormTransporters.fbFormTransporterBeforeScrewer.eState = E_Station.eReady OR P15_FormTransporters.fbFormTransporterBeforeScrewer.eState = E_Station.eManualMovement OR P15_FormTransporters.fbFormTransporterBeforeScrewer.eState = E_Station.eDisabled)
				;	

//Stacje sa w manualu albo w błędzie 
bStationsAreManualOrError := 
				(P01_BottleFeeder.fbBottleFeeder.eState = E_Station.eError OR P01_BottleFeeder.fbBottleFeeder.eState = E_Station.eManualMovement OR P01_BottleFeeder.fbBottleFeeder.eState = E_Station.eDisabled ) AND
				(P01_BottleFeeder.fbTurnTable.eState = E_Station.eError OR P01_BottleFeeder.fbTurnTable.eState = E_Station.eManualMovement OR P01_BottleFeeder.fbTurnTable.eState = E_Station.eDisabled) AND
				(P01_PucksInserter.fbPucksInserter.eState = E_Station.eError OR P01_PucksInserter.fbPucksInserter.eState = E_Station.eManualMovement OR P01_PucksInserter.fbPucksInserter.eState = E_Station.eDisabled) AND
				(P01_PucksInserter.fbTurnTable.eState = E_Station.eError OR P01_PucksInserter.fbTurnTable.eState = E_Station.eManualMovement OR P01_PucksInserter.fbTurnTable.eState = E_Station.eDisabled) AND
				(stBottleSorterRead.ePackMLAutoState = E_PMLState.ePMLState_RESETTING OR stBottleSorterRead.ePackMLAutoState = E_PMLState.ePMLState_IDLE OR NOT stBottleSorterRead.bEnable OR bBottleSorterDisable)  AND
				(P02_Dispencers.fbDispencersDragRightStation.eState = E_Station.eError OR P02_Dispencers.fbDispencersDragRightStation.eState = E_Station.eManualMovement OR P02_Dispencers.fbDispencersDragRightStation.eState = E_Station.eDisabled) AND 
				(P02_Dispencers.fbDispencersDragLeftStation.eState = E_Station.eError OR P02_Dispencers.fbDispencersDragLeftStation.eState = E_Station.eManualMovement OR P02_Dispencers.fbDispencersDragLeftStation.eState = E_Station.eDisabled) AND 
                (P02_Dispencers.fbDispencer1.eState = E_Station.eError OR P02_Dispencers.fbDispencer1.eState = E_Station.eManualMovement OR P02_Dispencers.fbDispencer1.eState = E_Station.eDisabled) AND
                (P02_Dispencers.fbDispencer2.eState = E_Station.eError OR P02_Dispencers.fbDispencer2.eState = E_Station.eManualMovement OR P02_Dispencers.fbDispencer2.eState = E_Station.eDisabled) AND
                (P02_Dispencers.fbDispencer3.eState = E_Station.eError OR P02_Dispencers.fbDispencer3.eState = E_Station.eManualMovement OR P02_Dispencers.fbDispencer3.eState = E_Station.eDisabled) AND
                (P02_Dispencers.fbDispencer4.eState = E_Station.eError OR P02_Dispencers.fbDispencer4.eState = E_Station.eManualMovement OR P02_Dispencers.fbDispencer4.eState = E_Station.eDisabled) AND
                (P02_Dispencers.fbDispencersCatch1Station.eState = E_Station.eError OR P02_Dispencers.fbDispencersCatch1Station.eState = E_Station.eManualMovement OR P02_Dispencers.fbDispencersCatch1Station.eState = E_Station.eDisabled) AND
                (P02_Dispencers.fbDispencersCatch2Station.eState = E_Station.eError OR P02_Dispencers.fbDispencersCatch2Station.eState = E_Station.eManualMovement OR P02_Dispencers.fbDispencersCatch2Station.eState = E_Station.eDisabled) AND
                (P02_Dispencers.fbDispencersCatch3Station.eState = E_Station.eError OR P02_Dispencers.fbDispencersCatch3Station.eState = E_Station.eManualMovement OR P02_Dispencers.fbDispencersCatch3Station.eState = E_Station.eDisabled) AND
                (P02_Dispencers.fbDispencersCatch4Station.eState = E_Station.eError OR P02_Dispencers.fbDispencersCatch4Station.eState = E_Station.eManualMovement OR P02_Dispencers.fbDispencersCatch4Station.eState = E_Station.eDisabled) AND
				(P05_Weight.fbWeight1.eState = E_Station.eError OR P05_Weight.fbWeight1.eState = E_Station.eManualMovement OR P05_Weight.fbWeight1.eState = E_Station.eDisabled) AND
    			(P05_Weight.fbWeight2.eState = E_Station.eError OR P05_Weight.fbWeight2.eState = E_Station.eManualMovement OR P05_Weight.fbWeight2.eState = E_Station.eDisabled) AND
				(P05_Weight.fbWeight3.eState = E_Station.eError OR P05_Weight.fbWeight3.eState = E_Station.eManualMovement OR P05_Weight.fbWeight3.eState = E_Station.eDisabled) AND
				(P05_Weight.fbWeight4.eState = E_Station.eError OR P05_Weight.fbWeight4.eState = E_Station.eManualMovement OR P05_Weight.fbWeight4.eState = E_Station.eDisabled) AND
				(P05_Weight.fbWeight5.eState = E_Station.eError OR P05_Weight.fbWeight5.eState = E_Station.eManualMovement OR P05_Weight.fbWeight5.eState = E_Station.eDisabled) AND
				(P05_Weight.fbWeight6.eState = E_Station.eError OR P05_Weight.fbWeight6.eState = E_Station.eManualMovement OR P05_Weight.fbWeight6.eState = E_Station.eDisabled) AND				
				(P05_Weight.fbWeightStation.eState = E_Station.eError OR P05_Weight.fbWeightStation.eState = E_Station.eManualMovement OR P05_Weight.fbWeightStation.eState = E_Station.eDisabled) AND
				(P05_Weight.fbWeightStation2Phase.eState = E_Station.eError OR P05_Weight.fbWeightStation2Phase.eState = E_Station.eManualMovement OR P05_Weight.fbWeightStation2Phase.eState = E_Station.eDisabled) AND
				(P06_LidFeeder.fbLidFeeder.eState = E_Station.eError OR P06_LidFeeder.fbLidFeeder.eState = E_Station.eManualMovement OR P06_LidFeeder.fbLidFeeder.eState = E_Station.eDisabled) AND 
				(P06_LidFeeder.fbLidFeeder2.eState = E_Station.eError OR P06_LidFeeder.fbLidFeeder2.eState = E_Station.eManualMovement OR P06_LidFeeder.fbLidFeeder2.eState = E_Station.eDisabled) AND
				(P06_LidFeeder.fbLidFeederDragStation.eState = E_Station.eError OR P06_LidFeeder.fbLidFeederDragStation.eState = E_Station.eManualMovement OR P06_LidFeeder.fbLidFeederDragStation.eState = E_Station.eDisabled) AND
				//(P06_LidPuttedCheck.fbLidPuttedCheck.eState = E_Station.eError OR P06_LidPuttedCheck.fbLidPuttedCheck.eState = E_Station.eManualMovement OR P06_LidPuttedCheck.fbLidPuttedCheck.eState = E_Station.eDisabled) AND 
				(P06_LidSealer.fbLidSealer.eState = E_Station.eError OR P06_LidSealer.fbLidSealer.eState = E_Station.eManualMovement OR P06_LidSealer.fbLidSealer.eState = E_Station.eDisabled) AND 
				(P06_LidSealer.fbLidSealer2.eState = E_Station.eError OR P06_LidSealer.fbLidSealer2.eState = E_Station.eManualMovement OR P06_LidSealer.fbLidSealer2.eState = E_Station.eDisabled) AND
				(P06_LidSealer.fbLidSealerDragStation.eState = E_Station.eError OR P06_LidSealer.fbLidSealerDragStation.eState = E_Station.eManualMovement OR P06_LidSealer.fbLidSealerDragStation.eState = E_Station.eDisabled) AND

				(P06_WickFeeder.fbWickFeederSt.eState = E_Station.eError OR P06_WickFeeder.fbWickFeederSt.eState = E_Station.eManualMovement OR P06_WickFeeder.fbWickFeederSt.eState = E_Station.eDisabled) AND
				(P06_WickFeeder.fbWickFeederDragStation.eState = E_Station.eError OR P06_WickFeeder.fbWickFeederDragStation.eState = E_Station.eManualMovement OR P06_WickFeeder.fbWickFeederDragStation.eState = E_Station.eDisabled) AND
				
				(P07_ROPP.fbROPPFeeder.eState = E_Station.eError OR P07_ROPP.fbROPPFeeder.eState = E_Station.eManualMovement OR P07_ROPP.fbROPPFeeder.eState = E_Station.eDisabled) AND
				(P07_ROPP.fbROPPDrag.eState = E_Station.eError OR P07_ROPP.fbROPPDrag.eState = E_Station.eManualMovement OR P07_ROPP.fbROPPDrag.eState = E_Station.eDisabled) AND
				(P07_ROPP.fbROPPCapping.eState = E_Station.eError OR P07_ROPP.fbROPPCapping.eState = E_Station.eManualMovement OR P07_ROPP.fbROPPCapping.eState = E_Station.eDisabled) AND

				(P08_CapFeeder.fbCapFeeder.eState = E_Station.eError OR P08_CapFeeder.fbCapFeeder.eState = E_Station.eManualMovement OR P08_CapFeeder.fbCapFeeder.eState = E_Station.eDisabled) AND
				(P08_CapSorter.fbCapSorterDragStation.eState = E_Station.eError OR P08_CapSorter.fbCapSorterDragStation.eState = E_Station.eManualMovement OR P08_CapSorter.fbCapSorterDragStation.eState = E_Station.eDisabled) AND				
				(stCapSorterRead.ePackMLAutoState = E_PMLState.ePMLState_RESETTING OR stCapSorterRead.ePackMLAutoState = E_PMLState.ePMLState_IDLE OR NOT stCapSorterRead.bEnable OR bCapSorterDisable)  AND				
				(P09_CapPuttedCheck.fbCapPuttedCheck.eState = E_Station.eError OR P09_CapPuttedCheck.fbCapPuttedCheck.eState = E_Station.eManualMovement OR P09_CapPuttedCheck.fbCapPuttedCheck.eState = E_Station.eDisabled) AND
   				(P10_GripperScrewer.fbGripperScrewersDragStation.eState = E_Station.eError OR P10_GripperScrewer.fbGripperScrewersDragStation.eState = E_Station.eManualMovement OR P10_GripperScrewer.fbGripperScrewersDragStation.eState = E_Station.eDisabled) AND
   	   			(P10_GripperScrewer.fbGripperScrewer1CatchStation.eState = E_Station.eError OR P10_GripperScrewer.fbGripperScrewer1CatchStation.eState = E_Station.eManualMovement OR P10_GripperScrewer.fbGripperScrewer1CatchStation.eState = E_Station.eDisabled) AND
				(P10_GripperScrewer.fbGripperScrewer2CatchStation.eState = E_Station.eError OR P10_GripperScrewer.fbGripperScrewer2CatchStation.eState = E_Station.eManualMovement OR P10_GripperScrewer.fbGripperScrewer2CatchStation.eState = E_Station.eDisabled) AND
    			(P11_CapCorrectCheck.fbCapCorrectCheck.eState = E_Station.eError OR P11_CapCorrectCheck.fbCapCorrectCheck.eState = E_Station.eManualMovement OR P11_CapCorrectCheck.fbCapCorrectCheck.eState = E_Station.eDisabled) AND
				(P13_BottleTransfer.fbBottleTransfer.eState = E_Station.eError OR P13_BottleTransfer.fbBottleTransfer.eState = E_Station.eManualMovement OR P13_BottleTransfer.fbBottleTransfer.eState = E_Station.eDisabled) AND 
				(P15_FormTransporters.fbFormTransporterDispencer.eState = E_Station.eError OR P15_FormTransporters.fbFormTransporterDispencer.eState = E_Station.eManualMovement OR P15_FormTransporters.fbFormTransporterDispencer.eState = E_Station.eDisabled) AND
				(P15_FormTransporters.fbFormTransporterScrewer.eState = E_Station.eError OR P15_FormTransporters.fbFormTransporterScrewer.eState = E_Station.eManualMovement OR P15_FormTransporters.fbFormTransporterScrewer.eState = E_Station.eDisabled) AND
 				(P15_FormTransporters.fbFormTransporterROPP.eState = E_Station.eError OR P15_FormTransporters.fbFormTransporterROPP.eState = E_Station.eManualMovement OR P15_FormTransporters.fbFormTransporterROPP.eState = E_Station.eDisabled) AND
				(P15_FormTransporters.fbFormTransporterBeforeScrewer.eState = E_Station.eError OR P15_FormTransporters.fbFormTransporterBeforeScrewer.eState = E_Station.eManualMovement OR P15_FormTransporters.fbFormTransporterBeforeScrewer.eState = E_Station.eDisabled)
				;	
							   

//Stacje sa gotowe albo w błędzie
bStationsAreReadyOrError :=
				(P01_BottleFeeder.fbBottleFeeder.eState = E_Station.eError OR P01_BottleFeeder.fbBottleFeeder.eState = E_Station.eReady OR P01_BottleFeeder.fbBottleFeeder.eState = E_Station.eDisabled ) AND
				(P01_BottleFeeder.fbTurnTable.eState = E_Station.eError OR P01_BottleFeeder.fbTurnTable.eState = E_Station.eReady OR P01_BottleFeeder.fbTurnTable.eState = E_Station.eDisabled) AND
				(P01_PucksInserter.fbPucksInserter.eState = E_Station.eError OR P01_PucksInserter.fbPucksInserter.eState = E_Station.eReady OR P01_PucksInserter.fbPucksInserter.eState = E_Station.eDisabled ) AND
				(P01_PucksInserter.fbTurnTable.eState = E_Station.eError OR P01_PucksInserter.fbTurnTable.eState = E_Station.eReady OR P01_PucksInserter.fbTurnTable.eState = E_Station.eDisabled) AND
				(stBottleSorterRead.ePackMLAutoState = E_PMLState.ePMLState_RESETTING OR stBottleSorterRead.ePackMLAutoState = E_PMLState.ePMLState_IDLE OR NOT stBottleSorterRead.bEnable OR bBottleSorterDisable)  AND
				(P02_Dispencers.fbDispencersDragRightStation.eState = E_Station.eError OR P02_Dispencers.fbDispencersDragRightStation.eState = E_Station.eReady OR P02_Dispencers.fbDispencersDragRightStation.eState = E_Station.eDisabled) AND 
				(P02_Dispencers.fbDispencersDragLeftStation.eState = E_Station.eError OR P02_Dispencers.fbDispencersDragLeftStation.eState = E_Station.eReady OR P02_Dispencers.fbDispencersDragLeftStation.eState = E_Station.eDisabled) AND 
                (P02_Dispencers.fbDispencer1.eState = E_Station.eError OR P02_Dispencers.fbDispencer1.eState = E_Station.eReady OR P02_Dispencers.fbDispencer1.eState = E_Station.eDisabled) AND
                (P02_Dispencers.fbDispencer2.eState = E_Station.eError OR P02_Dispencers.fbDispencer2.eState = E_Station.eReady OR P02_Dispencers.fbDispencer2.eState = E_Station.eDisabled) AND
                (P02_Dispencers.fbDispencer3.eState = E_Station.eError OR P02_Dispencers.fbDispencer3.eState = E_Station.eReady OR P02_Dispencers.fbDispencer3.eState = E_Station.eDisabled) AND
                (P02_Dispencers.fbDispencer4.eState = E_Station.eError OR P02_Dispencers.fbDispencer4.eState = E_Station.eReady OR P02_Dispencers.fbDispencer4.eState = E_Station.eDisabled) AND
                (P02_Dispencers.fbDispencersCatch1Station.eState = E_Station.eError OR P02_Dispencers.fbDispencersCatch1Station.eState = E_Station.eReady OR P02_Dispencers.fbDispencersCatch1Station.eState = E_Station.eDisabled) AND
                (P02_Dispencers.fbDispencersCatch2Station.eState = E_Station.eError OR P02_Dispencers.fbDispencersCatch2Station.eState = E_Station.eReady OR P02_Dispencers.fbDispencersCatch2Station.eState = E_Station.eDisabled) AND
                (P02_Dispencers.fbDispencersCatch3Station.eState = E_Station.eError OR P02_Dispencers.fbDispencersCatch3Station.eState = E_Station.eReady OR P02_Dispencers.fbDispencersCatch3Station.eState = E_Station.eDisabled) AND
                (P02_Dispencers.fbDispencersCatch4Station.eState = E_Station.eError OR P02_Dispencers.fbDispencersCatch4Station.eState = E_Station.eReady OR P02_Dispencers.fbDispencersCatch4Station.eState = E_Station.eDisabled) AND
				(P05_Weight.fbWeight1.eState = E_Station.eError OR P05_Weight.fbWeight1.eState = E_Station.eReady OR P05_Weight.fbWeight1.eState = E_Station.eDisabled) AND
    			(P05_Weight.fbWeight2.eState = E_Station.eError OR P05_Weight.fbWeight2.eState = E_Station.eReady OR P05_Weight.fbWeight2.eState = E_Station.eDisabled) AND
				(P05_Weight.fbWeight3.eState = E_Station.eError OR P05_Weight.fbWeight3.eState = E_Station.eReady OR P05_Weight.fbWeight3.eState = E_Station.eDisabled) AND
				(P05_Weight.fbWeight4.eState = E_Station.eError OR P05_Weight.fbWeight4.eState = E_Station.eReady OR P05_Weight.fbWeight4.eState = E_Station.eDisabled) AND
				(P05_Weight.fbWeight5.eState = E_Station.eError OR P05_Weight.fbWeight5.eState = E_Station.eReady OR P05_Weight.fbWeight5.eState = E_Station.eDisabled) AND
				(P05_Weight.fbWeight6.eState = E_Station.eError OR P05_Weight.fbWeight6.eState = E_Station.eReady OR P05_Weight.fbWeight6.eState = E_Station.eDisabled) AND				
				(P05_Weight.fbWeightStation.eState = E_Station.eError OR P05_Weight.fbWeightStation.eState = E_Station.eReady OR P05_Weight.fbWeightStation.eState = E_Station.eDisabled) AND
				(P05_Weight.fbWeightStation2Phase.eState = E_Station.eError OR P05_Weight.fbWeightStation2Phase.eState = E_Station.eReady OR P05_Weight.fbWeightStation2Phase.eState = E_Station.eDisabled) AND
				(P06_LidFeeder.fbLidFeeder.eState = E_Station.eError OR P06_LidFeeder.fbLidFeeder.eState = E_Station.eReady OR P06_LidFeeder.fbLidFeeder.eState = E_Station.eDisabled) AND 
				(P06_LidFeeder.fbLidFeeder2.eState = E_Station.eError OR P06_LidFeeder.fbLidFeeder2.eState = E_Station.eReady OR P06_LidFeeder.fbLidFeeder2.eState = E_Station.eDisabled) AND
				(P06_LidFeeder.fbLidFeederDragStation.eState = E_Station.eError OR P06_LidFeeder.fbLidFeederDragStation.eState = E_Station.eReady OR P06_LidFeeder.fbLidFeederDragStation.eState = E_Station.eDisabled) AND
				//(P06_LidPuttedCheck.fbLidPuttedCheck.eState = E_Station.eError OR P06_LidPuttedCheck.fbLidPuttedCheck.eState = E_Station.eReady OR P06_LidPuttedCheck.fbLidPuttedCheck.eState = E_Station.eDisabled) AND 
				(P06_LidSealer.fbLidSealer.eState = E_Station.eError OR P06_LidSealer.fbLidSealer.eState = E_Station.eReady OR P06_LidSealer.fbLidSealer.eState = E_Station.eDisabled) AND 
				(P06_LidSealer.fbLidSealer2.eState = E_Station.eError OR P06_LidSealer.fbLidSealer2.eState = E_Station.eReady OR P06_LidSealer.fbLidSealer2.eState = E_Station.eDisabled) AND
				(P06_LidSealer.fbLidSealerDragStation.eState = E_Station.eError OR P06_LidSealer.fbLidSealerDragStation.eState = E_Station.eReady OR P06_LidSealer.fbLidSealerDragStation.eState = E_Station.eDisabled) AND
				
				(P06_WickFeeder.fbWickFeederSt.eState = E_Station.eError OR P06_WickFeeder.fbWickFeederSt.eState = E_Station.eReady OR P06_WickFeeder.fbWickFeederSt.eState = E_Station.eDisabled) AND
				(P06_WickFeeder.fbWickFeederDragStation.eState = E_Station.eError OR P06_WickFeeder.fbWickFeederDragStation.eState = E_Station.eReady OR P06_WickFeeder.fbWickFeederDragStation.eState = E_Station.eDisabled) AND

				(P07_ROPP.fbROPPFeeder.eState = E_Station.eError OR P07_ROPP.fbROPPFeeder.eState = E_Station.eReady OR P07_ROPP.fbROPPFeeder.eState = E_Station.eDisabled) AND
				(P07_ROPP.fbROPPDrag.eState = E_Station.eError OR P07_ROPP.fbROPPDrag.eState = E_Station.eReady OR P07_ROPP.fbROPPDrag.eState = E_Station.eDisabled) AND
				(P07_ROPP.fbROPPCapping.eState = E_Station.eError OR P07_ROPP.fbROPPCapping.eState = E_Station.eReady OR P07_ROPP.fbROPPCapping.eState = E_Station.eDisabled) AND

				(P08_CapFeeder.fbCapFeeder.eState = E_Station.eError OR P08_CapFeeder.fbCapFeeder.eState = E_Station.eReady OR P08_CapFeeder.fbCapFeeder.eState = E_Station.eDisabled) AND
				(P08_CapSorter.fbCapSorterDragStation.eState = E_Station.eError OR P08_CapSorter.fbCapSorterDragStation.eState = E_Station.eReady OR P08_CapSorter.fbCapSorterDragStation.eState = E_Station.eDisabled) AND				
				(stCapSorterRead.ePackMLAutoState = E_PMLState.ePMLState_RESETTING OR stCapSorterRead.ePackMLAutoState = E_PMLState.ePMLState_IDLE OR NOT stCapSorterRead.bEnable OR bCapSorterDisable)  AND				
				(P09_CapPuttedCheck.fbCapPuttedCheck.eState = E_Station.eError OR P09_CapPuttedCheck.fbCapPuttedCheck.eState = E_Station.eReady OR P09_CapPuttedCheck.fbCapPuttedCheck.eState = E_Station.eDisabled) AND
   				(P10_GripperScrewer.fbGripperScrewersDragStation.eState = E_Station.eError OR P10_GripperScrewer.fbGripperScrewersDragStation.eState = E_Station.eReady OR P10_GripperScrewer.fbGripperScrewersDragStation.eState = E_Station.eDisabled) AND
   	   			(P10_GripperScrewer.fbGripperScrewer1CatchStation.eState = E_Station.eError OR P10_GripperScrewer.fbGripperScrewer1CatchStation.eState = E_Station.eReady OR P10_GripperScrewer.fbGripperScrewer1CatchStation.eState = E_Station.eDisabled) AND
				(P10_GripperScrewer.fbGripperScrewer2CatchStation.eState = E_Station.eError OR P10_GripperScrewer.fbGripperScrewer2CatchStation.eState = E_Station.eReady OR P10_GripperScrewer.fbGripperScrewer2CatchStation.eState = E_Station.eDisabled) AND
    			(P11_CapCorrectCheck.fbCapCorrectCheck.eState = E_Station.eError OR P11_CapCorrectCheck.fbCapCorrectCheck.eState = E_Station.eReady OR P11_CapCorrectCheck.fbCapCorrectCheck.eState = E_Station.eDisabled) AND
				(P13_BottleTransfer.fbBottleTransfer.eState = E_Station.eError OR P13_BottleTransfer.fbBottleTransfer.eState = E_Station.eReady OR P13_BottleTransfer.fbBottleTransfer.eState = E_Station.eDisabled) AND 
				(P15_FormTransporters.fbFormTransporterDispencer.eState = E_Station.eError OR P15_FormTransporters.fbFormTransporterDispencer.eState = E_Station.eReady OR P15_FormTransporters.fbFormTransporterDispencer.eState = E_Station.eDisabled) AND
				(P15_FormTransporters.fbFormTransporterScrewer.eState = E_Station.eError OR P15_FormTransporters.fbFormTransporterScrewer.eState = E_Station.eReady OR P15_FormTransporters.fbFormTransporterScrewer.eState = E_Station.eDisabled) AND
 				(P15_FormTransporters.fbFormTransporterROPP.eState = E_Station.eError OR P15_FormTransporters.fbFormTransporterROPP.eState = E_Station.eReady OR P15_FormTransporters.fbFormTransporterROPP.eState = E_Station.eDisabled) AND
				(P15_FormTransporters.fbFormTransporterBeforeScrewer.eState = E_Station.eError OR P15_FormTransporters.fbFormTransporterBeforeScrewer.eState = E_Station.eReady OR P15_FormTransporters.fbFormTransporterBeforeScrewer.eState = E_Station.eDisabled)
				;	

fbIbDispencerAfterCheckFormSensor(bIn:=P02_Dispencers.IbDispencerAfterCheckFormSensor, 			tFilterTimeOn:=T#200MS, tFilterTimeOff:=T#200MS);
fbIbDispencer12NoColisionWhenDosingSensor	(bIn:=P02_Dispencers.IbDispencer12NoColisionWhenDosingSensor, 	tFilterTimeOn:=T#40MS, tFilterTimeOff:=T#40MS);
fbIbDispencer34NoColisionWhenDosingSensor	(bIn:=P02_Dispencers.IbDispencer34NoColisionWhenDosingSensor, 	tFilterTimeOn:=T#40MS, tFilterTimeOff:=T#40MS);	

//PackML Commands -> Cap/Jar Unboxers
stBottleSorterWrite.sPackMLCommand.bAbort				:= fbPMLAuto.Abort;
stBottleSorterWrite.sPackMLCommand.bClear				:= fbPMLAuto.Clear;
sTBottleSorterWrite.sPackMLCommand.bComplete			:= fbPMLAuto.Complete;
stBottleSorterWrite.sPackMLCommand.bHold				:= fbPMLAuto.Hold;
stBottleSorterWrite.sPackMLCommand.bReset				:= fbPMLAuto.Reset;
stBottleSorterWrite.sPackMLCommand.bStart				:= fbPMLAuto.Start;
stBottleSorterWrite.sPackMLCommand.bStateComplete		:= fbPMLAuto.StateComplete;
stBottleSorterWrite.sPackMLCommand.bStop				:= fbPMLAuto.Stop;
stBottleSorterWrite.sPackMLCommand.bSuspend				:= fbPMLAuto.Suspend;
stBottleSorterWrite.sPackMLCommand.bUnHold				:= fbPMLAuto.UnHold; 


stCapSorterWrite.sPackMLCommand.bAbort					:= fbPMLAuto.Abort;
stCapSorterWrite.sPackMLCommand.bClear					:= fbPMLAuto.Clear;
stCapSorterWrite.sPackMLCommand.bComplete				:= fbPMLAuto.Complete;
stCapSorterWrite.sPackMLCommand.bHold					:= fbPMLAuto.Hold;
stCapSorterWrite.sPackMLCommand.bReset					:= fbPMLAuto.Reset;
stCapSorterWrite.sPackMLCommand.bStart					:= fbPMLAuto.Start;
stCapSorterWrite.sPackMLCommand.bStateComplete			:= fbPMLAuto.StateComplete;
stCapSorterWrite.sPackMLCommand.bStop					:= fbPMLAuto.Stop;
stCapSorterWrite.sPackMLCommand.bSuspend				:= fbPMLAuto.Suspend;
stCapSorterWrite.sPackMLCommand.bUnHold					:= fbPMLAuto.UnHold;

//Drag
ftbFormsDragingLeftRun	(CLK:=	P02_Dispencers.fbDispencersDragLeftStation.bCycleDone (*VIS.bFormsDragingLeftRun*),	Q=>); 
rtbFormsDragingLeftRun	(CLK:=	VIS.bFormsDragingLeftRun,	Q=>); 
rtbFormsDragingRightRun	(CLK:=	VIS.bFormsDragingRightRun,	Q=>); 
ftbFormsDragingRightRun	(CLK:=	P02_Dispencers.fbDispencersDragRightStation.bCycleDone (*VIS.bFormsDragingRightRun*),	Q=>);
END_ACTION

ACTION ACT_SignalsFormsCounting:
//Czujnik miedzy wagami a zakrecarka
P08_CapSorter.IbCapSorterGateScrewerSensor; // 13formatek na tym czujniku // Czujnik blizej zakrecarek
P08_CapSorter.IbCapSorterGateWeightSensor; // Czujnik kolejki blizej wag
fbIbCapSorterGateScrewerSensor	(bIn:=P08_CapSorter.IbCapSorterGateScrewerSensor,		tFilterTimeon:=T#100MS, tFilterTimeOff:=T#1000MS); 
fbIbCapSorterGateWeightSensor	(bIn:=P08_CapSorter.IbCapSorterGateWeightSensor OR MAIN.IbLidSealerAfterSensor,		tFilterTimeon:=T#4000MS, tFilterTimeOff:=T#500MS); //bylo 2000 i 1000
fbIbCapCorrectCheckFormSensor	(bIn:=P11_CapCorrectCheck.IbCapCorrectCheckFormSensor,	tFilterTimeon:=T#1000MS, tFilterTimeOff:=T#1000MS); 
	

//	Ilość formatek między wagą a sorterem nakrętek

//	Dozowniki w 1phase wypuszczają gdy 
//	(VIS.iNumbersOfFormsBetweenWeightAndScrewers <= 25 OR VIS.bWeight1EnableShow)

//	Waga wypuszcza gdy 
//	bCanReleaseForm	:= VIS.iNumbersOfFormsBetweenWeightAndScrewers <= 14;


//	Sorter nakrętek wypuszcza gdy
//	VIS.iNumbersOfFormsBetweenWeightAndScrewers>=8

(*
MAIN.ftfbFilteredCapSorterFormsSensorGate.Q; 
bCounterDisabled := FALSE;			

IF bCapSorterDisable THEN
	iSetNumbersOfFormsBetweenWeightAndScrewers	:=	17;
ELSE
	iSetNumbersOfFormsBetweenWeightAndScrewers	:=	25;
END_IF

   
IF tofTransportersWorking.Q THEN // dp Zmiana na ilośc formatek między zakręcarką a sorterem nasadek
	
	IF ftfbIbWeightFirstFormSensor.Q  OR ftfbIbWeightFirstForm2PhaseSensor.Q THEN
		VIS.iNumbersOfFormsBetweenWeightAndScrewers		:= VIS.iNumbersOfFormsBetweenWeightAndScrewers + 1;
	END_IF
	//IF ftfbIbCapPuttedCheckFormSensor.Q THEN
//	IF MAIN.ftfbFilteredCapSorterFormsSensorGate.Q THEN
//		VIS.iNumbersOfFormsBetweenWeightAndScrewers		:= VIS.iNumbersOfFormsBetweenWeightAndScrewers - 1;
//	END_IF
	IF ftfbIbCapPuttedCheckFormSensor.Q THEN
		VIS.iNumbersOfFormsBetweenWeightAndScrewers		:= VIS.iNumbersOfFormsBetweenWeightAndScrewers - 1;
	END_IF
	IF VIS.iNumbersOfFormsBetweenWeightAndScrewers<0 THEN
		VIS.iNumbersOfFormsBetweenWeightAndScrewers :=	0;
	END_IF
	
END_IF
*)
END_ACTION

ACTION ACT_SignalsLidFeeder:
fb2IbLidFeederThirdFormSensor		(bIn:=MAIN.IbLidFeederThirdFormSensor,	tFilterTimeOn:=T#1S500MS, tFilterTimeOff:=T#20MS);
fb2IbLidSealerSecondFormSensor		(bIn:=MAIN.IbLidSealerSecondFormSensor,	tFilterTimeOn:=T#1S, tFilterTimeOff:=T#20MS);
fbNotIbLidSealerSecondFormSensor	(bIn:=NOT MAIN.IbLidSealerSecondFormSensor,	tFilterTimeOn:=T#5S, tFilterTimeOff:=T#20MS);


tonbFormTransportersScrewerCmdStart (IN:=bFormTransportersScrewerCmdStart,	PT:=T#200MS);//dp
END_ACTION

ACTION ACT_SignalsROPP:


fbIbROPPSevenFormSensor				(bIN:=	P07_ROPP.IbROPPSevenFormSensor, tFilterTimeon:=T#100MS, tFilterTimeOff:=T#0MS); //bylo 190,0
fbIbROPPSevenFormSensor2			(bIN:=	P07_ROPP.IbROPPSevenFormSensor, tFilterTimeon:=T#30MS, tFilterTimeOff:=T#30MS); 
rtfbIbROPPSevenFormSensor2			(CLK:=	fbIbROPPSevenFormSensor2.bOUT,	Q=>);
ftfbIbROPPSevenFormSensor2			(CLK:=	fbIbROPPSevenFormSensor2.bOUT,	Q=>);

ftbReadedCardBeforeROPP				(CLK:=	P07_ROPP.bReadedCardBeforeROPP,	Q=>);
tonbReadedCardBeforeROPP			(IN:=	P07_ROPP.bReadedCardBeforeROPP,	PT:=T#2s);

fbIbROPPThirdFormSensor				(bIN:=	P07_ROPP.IbROPPThirdFormSensor, tFilterTimeon:=T#190MS, tFilterTimeOff:=T#30MS); //bylo 30 i 30

tonROPPThirdFormSensor				(IN:=	P07_ROPP.IbROPPThirdFormSensor (*AND (P15_FormTransporters.fbFormTransporterROPP.eState = eRunning)*),		PT:=T#200MS);//bylo 500 
tonROPPThirdFormSensor2				(IN:=	P07_ROPP.IbROPPThirdFormSensor ,	PT:=T#3S);//bylo 500

rtfbIbROPPThirdFormSensor			(CLK:=	fbIbROPPThirdFormSensor.bOut,	Q=>);
rtfbIbROPPThirdFormSensor2			(CLK:=	P07_ROPP.IbROPPThirdFormSensor ,Q=>);
ftfbIbROPPThirdFormSensor			(CLK:=	fbIbROPPThirdFormSensor.bOut,	Q=>);

tonROPPAfterFormSensor				(IN:=	(NOT P07_ROPP.IbROPPAfterFormSensor) AND (P15_FormTransporters.fbFormTransporterScrewerState.eState = eRunning) AND iROPPAfterFormCounter < 2 AND NOT VIS_ROPP.bROPPDragRun,	PT:=T#5S);
fbIbROPPAfterFormSensor				(bIn:=	P07_ROPP.IbROPPAfterFormSensor, tFilterTimeon:=T#35MS, tFilterTimeOff:=T#35MS); 
fbIbROPPAfterFormSensor2			(bIn:=	P07_ROPP.IbROPPAfterFormSensor, tFilterTimeon:=T#60MS, tFilterTimeOff:=T#60MS); 
fbIbROPPAfter3FormSensor			(bIn:=	P07_ROPP.IbROPPAfter3FormSensor, tFilterTimeon:=T#2S, tFilterTimeOff:=T#400MS); 

ftIbROPPAfterFormSensor				(CLK:=	fbIbROPPAfterFormSensor.bOut,	Q=>);

fbbReadedCardAfterROPP				(bIN:=	P07_ROPP.bReadedCardAfterROPP, tFilterTimeon:=T#0MS, tFilterTimeOff:=T#0MS); 
rtfbbReadedCardAfterROPP			(CLK:=	fbbReadedCardAfterROPP.bOUT,	Q=>);
ftfbbReadedCardAfterROPP			(CLK:=	fbbReadedCardAfterROPP.bOUT,	Q=>);

bROPPReady	:=		(NOT bROPPCappingEnable OR P07_ROPP.fbROPPCapping.eState = E_Station.eReady AND NOT P07_ROPP.fbROPPCapping.bRun1) AND
					(NOT bROPPCappingEnable OR P07_ROPP.fbROPPCapping.eState = E_Station.eReady AND NOT P07_ROPP.fbROPPCapping.bRun2) AND
					tonDelayAfterStart.Q;

fbROPPIbCapSorterBeforeFourthFormCheckFormSensor (bIN:=MAIN.IbCapSorterBeforeFourthFormCheckFormSensor, tFilterTimeon:=T#1.5S, tFilterTimeOff:=T#200MS); //bylo 3 s i 500 ms
END_ACTION

ACTION ACT_Statistics:


VIS.lrWeight1Mass;
VIS.lrWeight2Mass;
VIS.lrWeight3Mass;
VIS.lrWeight4Mass;
VIS.lrWeight5Mass;
VIS.lrWeight6Mass;
END_ACTION

ACTION ACT_Stopped:

// Wyjątek, przejście do bazownia z trybu manualnego
IF NOT bHomingDialog AND NOT (fbPMLModeManager.eModeStatus = Tc3_PackML.E_PMLUnitMode.ePMLUnitMode_MANUAL) THEN
	ACT_ResetCommands();
	iTestResetCommandsStopped	:=	iTestResetCommandsStopped	+	1; 
END_IF

//Brak błędów, przejście do Resetting
IF NOT VIS.bErrorOccure THEN
	fbPMLAuto.Reset					:= TRUE; 
	fbPMLManual.Reset				:= TRUE;
END_IF


(***************************)
IF tonResetErrorVisuCmd.Q THEN
	nResetErrorVisuCmd:=0;
END_IF
IF rtResetAlarmTrigger.Q THEN
	nResetErrorVisuCmd:=nResetErrorVisuCmd+1;
END_IF
IF nResetErrorVisuCmd > 2 THEN
	VIS.bResetErrorVisuCmd := TRUE;
END_IF

(***************************)
END_ACTION

ACTION ACT_Stopping:
ACT_PhaseChanging(); //Procedura zmiany fazy (jednofazowe-dwufazowe)
ACT_CycleLogic();
ACT_ResetCommandsHoming();


bStoppingWeight1 := (iWeightCase = 0 OR iWeightCase = 50 OR NOT GVL.bWeightLiftEnable OR P05_Weight.fbWeightStation.eState = E_Station.eError) ;
bStoppingWeight2 := (iWeightCase = 20 AND NOT P05_Weight.IbWeight1FormSensor AND NOT P05_Weight.IbWeight2FormSensor AND NOT P05_Weight.IbWeight3FormSensor AND NOT P05_Weight.IbWeight4FormSensor AND 
					NOT P05_Weight.IbWeight1ActuatorSensorUp AND NOT P05_Weight.IbWeight2ActuatorSensorUp AND NOT P05_Weight.IbWeight3ActuatorSensorUp AND NOT P05_Weight.IbWeight4ActuatorSensorUp);
		
